(* CODESYS project Discrete.library
   Placeholder: Discrete
   Title: Discrete
   Version: 2025.10.15.1
   Company: Photara

Project tree, tasks and I/O mapping:
  libraries: Base, * (Photara); Tc2_Standard, * (Beckhoff Automation GmbH); Tc2_System, * (Beckhoff Automation GmbH); TcUnit, * (www.tcunit.org)
  DUTs/
    data type E_DiscreteComponentState
    data type E_DiscretePositionType
    data type ST_DiscreteConfiguration
    data type ST_DiscreteStatus
  GVLs/
    global variables GC_Discrete
    global variables GPL_Discrete
  ITFs/
    interface I_DiscreteBase: Activate, Deactivate, P_DiscreteStatus
    interface I_DiscreteBaseConfiguration: P_DiscreteConfiguration
  POUs/
    Actuator/
      GVLs/
        global variables GC_Actuator
        global variables GPL_Actuator
      ITFs/
        interface I_ActuatorBase: Extend, Retract
      function block FB_Actuator [ST]: Extend, Retract, Activate, Deactivate, _SetCommandPermIntlkConfiguration, CyclicLogic
      function block FB_ActuatorFeedback [ST]: _EvaluateCompletionConditions, _InitializeChildrenDependencies, _SetDependencyConfiguration, CyclicLogic
    Tests/
      MockComponents/
        function block FB_TestActuator [ST]: P_TP_CmdConfigurations, P_TP_Commands, P_TP_iControlMode, P_TP_iSystemPermIntlk, P_TP_PermIntlkConfigurations, CyclicLogic
        function block FB_TestActuatorFeedback [ST]: P_I_SensorCfgExt, P_I_SensorCfgRet, P_I_SensorExt, P_I_SensorRet, _InitializeChildrenDependencies, _SetDependencyConfiguration, CyclicLogic
      function block FB_ActuatorBasicTests [ST]: _GetDiscreteComponent, _GetDiscreteComponentConfig
      function block FB_ActuatorFeedbackTests [ST]: _GetDiscreteComponent, _GetDiscreteComponentConfig, Test_FeedbackExtend_CompletesEarlyOnSensor, Test_FeedbackExtend_TimeoutWithoutSensor, Test_FeedbackRetract_CompletesEarlyOnSensor, Test_FeedbackRetract_TimeoutWithoutSensor
      function block FB_DiscreteBaseTests [ST]: _GetDiscreteComponent, _GetDiscreteComponentConfig, Test_ActivateCommandIdempotency, Test_CoilTruthTable_Active, Test_CoilTruthTable_Alternate, Test_CoilTruthTable_BothOn_FaultExpected, Test_CoilTruthTable_Neutral, Test_DeactivateCommandIdempotency, Test_DeviceReportsError_SetsFaultFlagAndOutputsOff, Test_DirectTransition_ActiveToAlternate, Test_DirectTransition_AlternateToActive, Test_ErrorRecovery_ClearsAndReturnsToNeutral, Test_InitializationSetsNeutralStateWithNoOutputs, Test_InvalidCommand_DoesNotChangeOutputs, Test_PermissiveInterlock_BlocksActivation, Test_PermissiveInterlock_BlocksAlternate, Test_RapidStateChanges_EndInExpectedState, Test_StateStabilityAcrossMultipleCycles, Test_ThreePositionDevice_ActivatesAlternateOutputOnly, Test_ThreePositionDevice_ActivatesPrimaryOutputOnly, Test_ThreePositionDevice_DeactivateTurnsOffBothOutputs, Test_ThreePositionDevice_NeverActivatesBothOutputsSimultaneously, Test_TransitionFromActiveToAlternateTurnsOffActiveFirst, Test_TwoPositionDevice_ActivatesCorrectOutput, Test_TwoPositionDevice_DeactivatesAllOutputs, Test_TwoPositionDevice_IgnoresAlternateRequest
      function block FB_ElectrostaticTests [ST]: _GetDiscreteComponent, _GetDiscreteComponentConfig
      function block FB_VacuumPurgeTests [ST]: _GetDiscreteComponent, _GetDiscreteComponentConfig
    function block FB_DiscreteBase [ST]: CyclicLogic, Activate, Deactivate, P_DiscreteConfiguration, P_DiscreteStatus, _InitializeReferences, _SetCommandPermIntlkConfiguration, _Activate, _Deactivate, _EvaluateCompletionConditions, _UpdateComponentStatus
    function block FB_Electrostatic [ST]: Activate, Deactivate, CyclicLogic
    function block FB_VacuumPurge [ST]: Activate, Deactivate, CyclicLogic, Purge, Vacuum
    program MAIN [ST]
    program PRG_TEST [ST]
*)

// DUTs/E_DiscreteComponentState
{attribute 'qualified_only'}
{attribute 'strict'}
{attribute 'to_string'}
TYPE E_DiscreteComponentState :
(
	Indeterminate := 0, //Undefined/Init
	Neutral 	:= 1, //Off/Determined but no output
	Active 		:= 2, //On/Vaccum
	Alternate	:= 3 //Purge
);
END_TYPE

// DUTs/E_DiscretePositionType
{attribute 'qualified_only'}
{attribute 'strict'}
{attribute 'to_string'}
TYPE E_DiscretePositionType  :
(
	TwoPositionDevice := 0,
	ThreePositionDevice := 1
);
END_TYPE

// DUTs/ST_DiscreteConfiguration
TYPE ST_DiscreteConfiguration :
STRUCT
	ComponentConfiguration 	: REFERENCE TO ST_ComponentConfiguration;
	PositionType			: E_DiscretePositionType;
	ActivationDuration		: TIME	:= Tc2_System.Global_Variables.DEFAULT_ADS_TIMEOUT; // assuming no feedback
	DeactivationDuration	: TIME 	:= T#10MS; // assuming no feedback
END_STRUCT
END_TYPE

// DUTs/ST_DiscreteStatus
TYPE ST_DiscreteStatus :
STRUCT
	ComponentStatus 		: REFERENCE TO ST_ComponentStatus;
	BinaryComponentState 	: E_DiscreteComponentState;
	
	PrimaryOutput 	AT %Q*	: BOOL; // ie., Vaccum
	SecondaryOutput	AT %Q*	: BOOL; // ie., Purge
END_STRUCT
END_TYPE

// GVLs/GC_Discrete
{attribute 'qualified_only'}
{attribute 'global_init_slot' := '40615'}
VAR_GLOBAL CONSTANT
	INDEX_COMMAND_MIN 	: DINT := GPL_Discrete.INDEX_COMMAND_MIN;
	INDEX_COMMAND_MAX 	: DINT := GPL_Discrete.INDEX_COMMAND_MAX;
	CMD_VAC				: DINT := 2;
	CMD_PURGE			: DINT := 3;
	CMD_EXTEND			: DINT := 4;
	CMD_RETRACT			: DINT := 5;
	INDEX_TEST_MIN		: DINT := 0;
	INDEX_TEST_MAX		: DINT := 30;
END_VAR

// GVLs/GPL_Discrete
{attribute 'qualified_only'}
{attribute 'global_init_slot' := '40515'}
VAR_GLOBAL CONSTANT
	INDEX_COMMAND_MIN 	: DINT := 0;
	INDEX_COMMAND_MAX 	: DINT := 4;
END_VAR

// POUs/Actuator/GVLs/GC_Actuator
{attribute 'qualified_only'}
{attribute 'global_init_slot' := '40603'}
VAR_GLOBAL CONSTANT
	INDEX_COMMAND_MIN		: DINT := GPL_Actuator.INDEX_COMMAND_MIN;
	INDEX_COMMAND_MAX		: DINT := GPL_Actuator.INDEX_COMMAND_MAX;
	Extend					: DINT := 2;
END_VAR

// POUs/Actuator/GVLs/GPL_Actuator
{attribute 'qualified_only'}
{attribute 'global_init_slot' := '40503'}
VAR_GLOBAL CONSTANT
	INDEX_COMMAND_MIN		: DINT := 0;
	INDEX_COMMAND_MAX		: DINT := 7;
END_VAR

// ITFs/I_DiscreteBase
INTERFACE I_DiscreteBase EXTENDS Base.I_BaseCyclic

METHOD Activate : Base.E_CommandResult
END_METHOD

METHOD Deactivate : Base.E_CommandResult
END_METHOD

PROPERTY P_DiscreteStatus : REFERENCE TO ST_DiscreteStatus
GET
END_GET
END_PROPERTY

END_INTERFACE

// ITFs/I_DiscreteBaseConfiguration
INTERFACE I_DiscreteBaseConfiguration EXTENDS Base.I_BaseCyclic

PROPERTY P_DiscreteConfiguration : REFERENCE TO ST_DiscreteConfiguration
GET
END_GET
END_PROPERTY

END_INTERFACE

// POUs/Actuator/ITFs/I_ActuatorBase
INTERFACE I_ActuatorBase EXTENDS __SYSTEM.IQueryInterface

METHOD Extend : E_CommandResult
VAR_INPUT
END_VAR
END_METHOD

METHOD Retract : E_CommandResult
VAR_INPUT
END_VAR
END_METHOD

END_INTERFACE

// POUs/Actuator/FB_Actuator
{attribute 'no_explicit_call' := 'do not call this POU directly'}
FUNCTION_BLOCK FB_Actuator EXTENDS FB_DiscreteBase IMPLEMENTS I_ActuatorBase
VAR CONSTANT
	// Use base class command indices - no need for separate actuator command indices
	// Extend = Activate (INDEX_CMD_ACTIVATE from base class)
	// Retract = Deactivate (INDEX_CMD_DEACTIVATE from base class)
END_VAR

VAR
	TestPermissiveFalse	: BOOL;
	TestPermissiveTrue	: BOOL := TRUE;
END_VAR

METHOD Extend : E_CommandResult
// Alias for Activate (Extend is the active state)
Extend := Activate();
END_METHOD

METHOD Retract : E_CommandResult
// Alias for Deactivate (Retract is the idle state)
Retract := Deactivate();
END_METHOD

METHOD Activate : Base.E_CommandResult
// Simply call the parent's Activate method - it handles everything
Activate := SUPER^.Activate();
END_METHOD

METHOD Deactivate : Base.E_CommandResult
// Simply call the parent's Deactivate method - it handles everything
Deactivate := SUPER^.Deactivate();
END_METHOD

METHOD PROTECTED _SetCommandPermIntlkConfiguration : BOOL
// Call parent configuration FIRST to set up base commands
SUPER^._SetCommandPermIntlkConfiguration();

//Configure as Two-Position Device
SUPER^.DiscreteComponentConfiguration.PositionType := E_DiscretePositionType.TwoPositionDevice;

//Command Extend
SUPER^.DiscreteComponentConfiguration.ActivationDuration	:= T#20S;
SUPER^.DiscreteComponentConfiguration.DeactivationDuration	:= T#5S;

// Override base command descriptions to use actuator terminology (Extend maps to Activate)
CommandPermIntlkConfiguration[INDEX_CMD_ACTIVATE].P_CommandConfiguration.CommandDescription					:= 'Extend';
CommandPermIntlkConfiguration[INDEX_CMD_ACTIVATE].P_CommandConfiguration.CommandIndex							:= INDEX_CMD_ACTIVATE;
CommandPermIntlkConfiguration[INDEX_CMD_ACTIVATE].P_CommandConfiguration.CommandPOUName						:= 'Extend';
CommandPermIntlkConfiguration[INDEX_CMD_ACTIVATE].P_CommandConfiguration.Priority								:= Base.E_CommandPriority.Priority_Normal;
CommandPermIntlkConfiguration[INDEX_CMD_ACTIVATE].P_CommandConfiguration.TimeoutTime							:= SUPER^.DiscreteComponentConfiguration.ActivationDuration;
CommandPermIntlkConfiguration[INDEX_CMD_ACTIVATE].P_CommandConfiguration.CompletionCondition					REF= SUPER^.CommandCompletionConditions[INDEX_CMD_ACTIVATE];

CommandPermIntlkConfiguration[INDEX_CMD_ACTIVATE].P_CommandConfiguration.PermIntlkConfiguration.PermIntlkObj[0].Condition		REF= TestPermissiveTrue;
CommandPermIntlkConfiguration[INDEX_CMD_ACTIVATE].P_CommandConfiguration.PermIntlkConfiguration.PermIntlkObj[0].Description	:= 'TestPermssiveFalse';
CommandPermIntlkConfiguration[INDEX_CMD_ACTIVATE].P_CommandConfiguration.PermIntlkConfiguration.PermIntlkObj[0].Index	:= 0;

//Command Retract
// Override base command descriptions to use actuator terminology (Retract maps to Deactivate)
CommandPermIntlkConfiguration[INDEX_CMD_DEACTIVATE].P_CommandConfiguration.CommandDescription					:= 'Retract';
CommandPermIntlkConfiguration[INDEX_CMD_DEACTIVATE].P_CommandConfiguration.CommandIndex						:= INDEX_CMD_DEACTIVATE;
CommandPermIntlkConfiguration[INDEX_CMD_DEACTIVATE].P_CommandConfiguration.CommandPOUName						:= 'Retract';
CommandPermIntlkConfiguration[INDEX_CMD_DEACTIVATE].P_CommandConfiguration.Priority							:= Base.E_CommandPriority.Priority_High;
CommandPermIntlkConfiguration[INDEX_CMD_DEACTIVATE].P_CommandConfiguration.TimeoutTime							:= SUPER^.DiscreteComponentConfiguration.DeactivationDuration;
CommandPermIntlkConfiguration[INDEX_CMD_DEACTIVATE].P_CommandConfiguration.CompletionCondition					REF= SUPER^.CommandCompletionConditions[INDEX_CMD_DEACTIVATE];

// CommandPermIntlkConfiguration[INDEX_COMMAND_RETRACT].P_CommandConfiguration.PermIntlkConfiguration.PermIntlkObj[].Condition	:= ;
// CommandPermIntlkConfiguration[INDEX_COMMAND_RETRACT].P_CommandConfiguration.PermIntlkConfiguration.PermIntlkObj[].Description	:= ;
// CommandPermIntlkConfiguration[INDEX_COMMAND_RETRACT].P_CommandConfiguration.PermIntlkConfiguration.PermIntlkObj[].Index	:= ;

_SetCommandPermIntlkConfiguration	:= TRUE;
END_METHOD

METHOD CyclicLogic
SUPER^.CyclicLogic();
END_METHOD

END_FUNCTION_BLOCK

// POUs/FB_DiscreteBase
{attribute 'no_explicit_call' := 'do not call this POU directly'}
FUNCTION_BLOCK ABSTRACT FB_DiscreteBase EXTENDS FB_Component<GC_Discrete.INDEX_COMMAND_MIN, GC_Discrete.INDEX_COMMAND_MAX> IMPLEMENTS I_DiscreteBase, I_DiscreteBaseConfiguration
VAR CONSTANT
	INDEX_CMD_ACTIVATE			: DINT := 0;
	INDEX_CMD_DEACTIVATE 		: DINT := 1;
END_VAR
VAR
	DiscreteComponentConfiguration				: ST_DiscreteConfiguration;
	DiscreteComponentStatus						: ST_DiscreteStatus;
END_VAR

METHOD CyclicLogic
SUPER^.CyclicLogic();
END_METHOD

METHOD Activate : Base.E_CommandResult
ExecuteCommand(CmdIndex := INDEX_CMD_ACTIVATE);

IF SUPER^.iCommands[INDEX_CMD_ACTIVATE].P_CommandStatus.Result = Base.E_CommandResult.Accepted THEN
	_Activate();
END_IF

Activate := SUPER^.iCommands[INDEX_CMD_ACTIVATE].P_CommandStatus.Result;
END_METHOD

METHOD Deactivate : Base.E_CommandResult
ExecuteCommand(CmdIndex := INDEX_CMD_DEACTIVATE);

IF SUPER^.iCommands[INDEX_CMD_DEACTIVATE].P_CommandStatus.Result = Base.E_CommandResult.Accepted THEN
	_Deactivate();
END_IF

Deactivate := SUPER^.iCommands[INDEX_CMD_DEACTIVATE].P_CommandStatus.Result;
END_METHOD

PROPERTY P_DiscreteConfiguration : REFERENCE TO ST_DiscreteConfiguration
GET
P_DiscreteConfiguration REF= DiscreteComponentConfiguration;
END_GET
END_PROPERTY

PROPERTY P_DiscreteStatus : REFERENCE TO ST_DiscreteStatus
GET
P_DiscreteStatus REF= DiscreteComponentStatus;
END_GET
END_PROPERTY

METHOD PROTECTED _InitializeReferences : BOOL
//Initialize data references
//Order is important!
BaseConfiguration.InstancePath 							REF= InstancePath;

ComponentConfiguration.BaseConfiguration 				REF= SUPER^.BaseConfiguration;
                                                    
ComponentStatus.BaseStatus								REF= SUPER^.BaseStatus;

ComponentStatus.AmsNetId								REF= ComponentConfiguration.AmsNetId;
                                                    
DiscreteComponentConfiguration.ComponentConfiguration	REF= SUPER^.ComponentConfiguration;

DiscreteComponentStatus.ComponentStatus					REF= SUPER^.ComponentStatus;

_InitializeReferences				:= TRUE;
END_METHOD

METHOD PROTECTED _SetCommandPermIntlkConfiguration : BOOL
//Command On
CommandPermIntlkConfiguration[INDEX_CMD_ACTIVATE].P_CommandConfiguration.AbortOnInterlockDrop					:= TRUE;
CommandPermIntlkConfiguration[INDEX_CMD_ACTIVATE].P_CommandConfiguration.CommandDescription						:= 'Activate';
CommandPermIntlkConfiguration[INDEX_CMD_ACTIVATE].P_CommandConfiguration.CommandIndex							:= INDEX_CMD_ACTIVATE;
CommandPermIntlkConfiguration[INDEX_CMD_ACTIVATE].P_CommandConfiguration.CommandPOUName							:= 'Activate';
//CommandPermIntlkConfiguration[INDEX_CMD_ACTIVATE].P_CommandConfiguration.PermIntlkConfiguredAsInterlock		:= TRUE;
CommandPermIntlkConfiguration[INDEX_CMD_ACTIVATE].P_CommandConfiguration.Priority								:= Base.E_CommandPriority.Priority_Normal;
CommandPermIntlkConfiguration[INDEX_CMD_ACTIVATE].P_CommandConfiguration.CompletionCondition					REF= SUPER^.CommandCompletionConditions[INDEX_CMD_ACTIVATE];
//CommandPermIntlkConfiguration[INDEX_CMD_ACTIVATE].P_CommandConfiguration.TimeoutTime							:= DiscreteComponentConfiguration.ActivationDuration;

// CommandPermIntlkConfiguration[INDEX_CMD_ACTIVATE].P_CommandConfiguration.PermIntlkConfiguration.PermIntlkObj[].Condition	:= ;
// CommandPermIntlkConfiguration[INDEX_CMD_ACTIVATE].P_CommandConfiguration.PermIntlkConfiguration.PermIntlkObj[].Description	:= ;
// CommandPermIntlkConfiguration[INDEX_CMD_ACTIVATE].P_CommandConfiguration.PermIntlkConfiguration.PermIntlkObj[].Index	:= ;

//Command Off
//CommandPermIntlkConfiguration[INDEX_CMD_DEACTIVATE].P_CommandConfiguration.AbortOnInterlockDrop				:= TRUE;
CommandPermIntlkConfiguration[INDEX_CMD_DEACTIVATE].P_CommandConfiguration.CommandDescription					:= 'Deactivate';
CommandPermIntlkConfiguration[INDEX_CMD_DEACTIVATE].P_CommandConfiguration.CommandIndex							:= INDEX_CMD_DEACTIVATE;
CommandPermIntlkConfiguration[INDEX_CMD_DEACTIVATE].P_CommandConfiguration.CommandPOUName						:= 'Deactivate';
//CommandPermIntlkConfiguration[INDEX_CMD_DEACTIVATE].P_CommandConfiguration.PermIntlkConfiguredAsInterlock		:= TRUE;
CommandPermIntlkConfiguration[INDEX_CMD_DEACTIVATE].P_CommandConfiguration.Priority								:= Base.E_CommandPriority.Priority_High;
CommandPermIntlkConfiguration[INDEX_CMD_DEACTIVATE].P_CommandConfiguration.TimeoutTime							:= DiscreteComponentConfiguration.DeactivationDuration;
CommandPermIntlkConfiguration[INDEX_CMD_DEACTIVATE].P_CommandConfiguration.CompletionCondition					REF= SUPER^.CommandCompletionConditions[INDEX_CMD_DEACTIVATE];
CommandPermIntlkConfiguration[INDEX_CMD_DEACTIVATE].P_CommandConfiguration.TimeoutTime							:= DiscreteComponentConfiguration.DeactivationDuration;

// CommandPermIntlkConfiguration[INDEX_CMD_DEACTIVATE].P_CommandConfiguration.PermIntlkConfiguration.PermIntlkObj[].Condition	:= ;
// CommandPermIntlkConfiguration[INDEX_CMD_DEACTIVATE].P_CommandConfiguration.PermIntlkConfiguration.PermIntlkObj[].Description	:= ;
// CommandPermIntlkConfiguration[INDEX_CMD_DEACTIVATE].P_CommandConfiguration.PermIntlkConfiguration.PermIntlkObj[].Index	:= ;

_SetCommandPermIntlkConfiguration	:= TRUE;
END_METHOD

METHOD PROTECTED _Activate
// Continuous mode: Hold output ON while command is busy
DiscreteComponentStatus.PrimaryOutput := TRUE;
DiscreteComponentStatus.SecondaryOutput := FALSE; // Safety: ensure alternate is off
END_METHOD

METHOD PROTECTED _Deactivate
// Continuous mode: Hold output OFF while command is busy
DiscreteComponentStatus.PrimaryOutput := FALSE;
DiscreteComponentStatus.SecondaryOutput := FALSE; // Safety: ensure alternate is off
END_METHOD

METHOD PROTECTED _EvaluateCompletionConditions : BOOL
// Set default completion conditions - commands complete immediately after output transition
// Derived classes can override to use different completion criteria (timeout, sensor feedback, etc.)
SUPER^.CommandCompletionConditions[INDEX_CMD_ACTIVATE]            		:= (DiscreteComponentStatus.PrimaryOutput AND NOT DiscreteComponentStatus.SecondaryOutput);
SUPER^.CommandCompletionConditions[INDEX_CMD_DEACTIVATE]            	:= (NOT DiscreteComponentStatus.PrimaryOutput AND NOT DiscreteComponentStatus.SecondaryOutput);

// Call generic logging implementation
_EvaluateCompletionConditions := TRUE;
END_METHOD

METHOD PROTECTED _UpdateComponentStatus: Base.I_ComponentFull
// Check configuration for device type
IF DiscreteComponentConfiguration.PositionType = E_DiscretePositionType.TwoPositionDevice THEN
	// Two-position device: Secondary output is always FALSE
	// Only two states are valid: Active and Neutral
	DiscreteComponentStatus.SecondaryOutput := FALSE;

	// Update state based on primary output only
	IF DiscreteComponentStatus.PrimaryOutput THEN
		// Primary output active = Active state
		DiscreteComponentStatus.BinaryComponentState := E_DiscreteComponentState.Active;
	ELSE
		// Primary output inactive = Neutral state
		DiscreteComponentStatus.BinaryComponentState := E_DiscreteComponentState.Neutral;
	END_IF
ELSE
	// Three-position device: Support all three states
	// Update component state based on primary and secondary outputs
	IF DiscreteComponentStatus.SecondaryOutput THEN
		// Secondary output active = Alternate state (e.g., Purge)
		DiscreteComponentStatus.BinaryComponentState := E_DiscreteComponentState.Alternate;
	ELSIF DiscreteComponentStatus.PrimaryOutput THEN
		// Primary output active, secondary inactive = Active state (e.g., Vacuum)
		DiscreteComponentStatus.BinaryComponentState := E_DiscreteComponentState.Active;
	ELSIF NOT DiscreteComponentStatus.PrimaryOutput AND NOT DiscreteComponentStatus.SecondaryOutput THEN
		// Both outputs inactive = Neutral state (Off)
		DiscreteComponentStatus.BinaryComponentState := E_DiscreteComponentState.Neutral;
	ELSE
		// Should not reach here, but if we do = Indeterminate
		DiscreteComponentStatus.BinaryComponentState := E_DiscreteComponentState.Indeterminate;
	END_IF
END_IF

_UpdateComponentStatus := THIS^;
END_METHOD

END_FUNCTION_BLOCK

// POUs/Actuator/FB_ActuatorFeedback
{attribute 'no_explicit_call' := 'do not call this POU directly'}
FUNCTION_BLOCK FB_ActuatorFeedback EXTENDS FB_Actuator
VAR
	SensorFeedbackExtended		: Base.FB_Debounce;
	SensorFeedbackRetracted		: Base.FB_Debounce;
	iDebounceExt				: Base.I_Debounce	:= SensorFeedbackExtended;
	iDebounceRet				: Base.I_Debounce	:= SensorFeedbackRetracted;
END_VAR

METHOD PROTECTED _EvaluateCompletionConditions : BOOL
// Set feedback-specific completion conditions - commands complete when sensors confirm position
IF iDebounceExt <> 0 THEN
	SUPER^.CommandCompletionConditions[INDEX_CMD_ACTIVATE]            	:= iDebounceExt.P_DebounceStatus.DebouncedSignal;
END_IF

IF iDebounceRet <> 0 THEN
	SUPER^.CommandCompletionConditions[INDEX_CMD_DEACTIVATE]            	:= iDebounceRet.P_DebounceStatus.DebouncedSignal;
END_IF

// Call base class logging method
_EvaluateCompletionConditions := TRUE;
END_METHOD

METHOD PROTECTED _InitializeChildrenDependencies : BOOL
// Initialize concrete configurations and wire directly to Commands
FOR CommandIndexCyclic := LOWER_BOUND(Commands,1) TO UPPER_BOUND(Commands,1) BY 1 DO

	// Inject configurations directly - TwinCAT auto-converts to interfaces
	Commands[CommandIndexCyclic].InjectConfigurations(
		iComponent := THIS^,
		iCommandConfiguration := CommandPermIntlkConfiguration[CommandIndexCyclic],
		iPermIntlkConfiguration := CommandPermIntlkConfiguration[CommandIndexCyclic]);
		
	CommandPermIntlkConfiguration[CommandIndexCyclic].Initialize();
	Commands[CommandIndexCyclic].Initialize();
END_FOR

CommandBuffer.Initialize();

fbHashDJB2_PouName.Initialize();
HashTablePouName.Initialize();

SensorFeedbackExtended.Initialize();
SensorFeedbackRetracted.Initialize();

HashTablePouName.InjectHashFunction(iHashFunction := iHashDJB2_PouName);

_InitializeChildrenDependencies := TRUE;
END_METHOD

METHOD PROTECTED _SetDependencyConfiguration : BOOL
SensorFeedbackExtended.P_DebounceConfiguration.BaseConfiguration.InSimulation	:= TRUE;
SensorFeedbackRetracted.P_DebounceConfiguration.BaseConfiguration.InSimulation	:= TRUE;
SensorFeedbackExtended.P_DebounceConfiguration.tOnDelay		:= T#50MS;
SensorFeedbackExtended.P_DebounceConfiguration.tOffDelay	:= T#50MS;

_SetDependencyConfiguration	:= TRUE;
END_METHOD

METHOD CyclicLogic
SUPER^.CyclicLogic();

SensorFeedbackExtended.CyclicLogic();
SensorFeedbackRetracted.CyclicLogic();
END_METHOD

END_FUNCTION_BLOCK

// POUs/Tests/MockComponents/FB_TestActuator
FUNCTION_BLOCK FB_TestActuator EXTENDS FB_Actuator
VAR_INPUT
END_VAR
VAR_OUTPUT
END_VAR
VAR
END_VAR

PROPERTY P_TP_CmdConfigurations : REFERENCE TO ARRAY[MinIndexComponentCmd..MaxIndexComponentCmd] OF FB_CmdPermIntlkConfiguration
GET
P_TP_CmdConfigurations REF= SUPER^.CommandPermIntlkConfiguration;
END_GET
END_PROPERTY

PROPERTY P_TP_Commands : REFERENCE TO ARRAY[MinIndexComponentCmd..MaxIndexComponentCmd] OF FB_Command
GET
P_TP_Commands REF= SUPER^.Commands;
END_GET
END_PROPERTY

PROPERTY P_TP_iControlMode : REFERENCE TO I_ControlMode
GET
P_TP_iControlMode REF= SUPER^._ControlMode;
END_GET
END_PROPERTY

PROPERTY P_TP_iSystemPermIntlk : REFERENCE TO I_PermIntlk
GET
P_TP_iSystemPermIntlk REF= SUPER^._SystemPermIntlk;
END_GET
END_PROPERTY

PROPERTY P_TP_PermIntlkConfigurations : REFERENCE TO ARRAY[MinIndexComponentCmd..MaxIndexComponentCmd] OF FB_CmdPermIntlkConfiguration
GET
P_TP_PermIntlkConfigurations REF= SUPER^.CommandPermIntlkConfiguration;
END_GET
END_PROPERTY

METHOD CyclicLogic
SUPER^.CyclicLogic();
END_METHOD

END_FUNCTION_BLOCK

// POUs/Tests/MockComponents/FB_TestActuatorFeedback
{attribute 'no_explicit_call' := 'do not call this POU directly'}
FUNCTION_BLOCK FB_TestActuatorFeedback EXTENDS FB_TestActuator
VAR
	SensorFeedbackExtended		: Base.FB_Debounce;
	SensorFeedbackRetracted		: Base.FB_Debounce;
	iDebounceExt				: Base.I_Debounce				:= SensorFeedbackExtended;
	iDebounceRet				: Base.I_Debounce				:= SensorFeedbackRetracted;
	iDebounceConfigExt			: Base.I_DebounceConfiguration	:= SensorFeedbackExtended;
	iDebounceConfigRet			: Base.I_DebounceConfiguration  := SensorFeedbackRetracted;
END_VAR

PROPERTY P_I_SensorCfgExt : REFERENCE TO Base.I_DebounceConfiguration
GET
P_I_SensorCfgExt REF= iDebounceConfigExt;
END_GET
END_PROPERTY

PROPERTY P_I_SensorCfgRet : REFERENCE TO Base.I_DebounceConfiguration
GET
P_I_SensorCfgRet REF= iDebounceConfigRet;
END_GET
END_PROPERTY

PROPERTY P_I_SensorExt : REFERENCE TO Base.I_Debounce
GET
P_I_SensorExt REF= iDebounceExt;
END_GET
END_PROPERTY

PROPERTY P_I_SensorRet : REFERENCE TO Base.I_Debounce
GET
P_I_SensorRet REF= iDebounceRet;
END_GET
END_PROPERTY

METHOD PROTECTED _InitializeChildrenDependencies : BOOL
// Initialize concrete configurations and wire directly to Commands
FOR CommandIndexCyclic := LOWER_BOUND(Commands,1) TO UPPER_BOUND(Commands,1) BY 1 DO

	// Inject configurations directly - TwinCAT auto-converts to interfaces
	Commands[CommandIndexCyclic].InjectConfigurations(
		iComponent := THIS^,
		iCommandConfiguration := CommandPermIntlkConfiguration[CommandIndexCyclic],
		iPermIntlkConfiguration := CommandPermIntlkConfiguration[CommandIndexCyclic]);
		
	CommandPermIntlkConfiguration[CommandIndexCyclic].Initialize();
	Commands[CommandIndexCyclic].Initialize();
END_FOR

CommandBuffer.Initialize();

fbHashDJB2_PouName.Initialize();
HashTablePouName.Initialize();

SensorFeedbackExtended.Initialize();
SensorFeedbackRetracted.Initialize();

HashTablePouName.InjectHashFunction(iHashFunction := iHashDJB2_PouName);

_InitializeChildrenDependencies := TRUE;
END_METHOD

METHOD PROTECTED _SetDependencyConfiguration : BOOL
SensorFeedbackExtended.P_DebounceConfiguration.BaseConfiguration.InSimulation	:= TRUE;
SensorFeedbackRetracted.P_DebounceConfiguration.BaseConfiguration.InSimulation	:= TRUE;
SensorFeedbackExtended.P_DebounceConfiguration.tOnDelay		:= T#50MS;
SensorFeedbackExtended.P_DebounceConfiguration.tOffDelay	:= T#50MS;

_SetDependencyConfiguration	:= TRUE;
END_METHOD

METHOD CyclicLogic
SUPER^.CyclicLogic();

SensorFeedbackExtended.CyclicLogic();
SensorFeedbackRetracted.CyclicLogic();
END_METHOD

END_FUNCTION_BLOCK

// POUs/Tests/FB_ActuatorBasicTests
FUNCTION_BLOCK FB_ActuatorBasicTests EXTENDS FB_DiscreteBaseTests

VAR
	afbActuator			: ARRAY[GC_Discrete.INDEX_TEST_MIN..GC_Discrete.INDEX_TEST_MAX] OF FB_TestActuator;
END_VAR

// All test methods are inherited from FB_DiscreteBaseTests
SUPER^();

METHOD PROTECTED _GetDiscreteComponent : I_DiscreteBase
VAR_INPUT
	Index : DINT;
END_VAR
// Return the actuator instance at the given index
_GetDiscreteComponent := afbActuator[Index];
END_METHOD

METHOD PROTECTED _GetDiscreteComponentConfig : I_DiscreteBaseConfiguration
VAR_INPUT
	Index : DINT;
END_VAR
// Return the actuator instance at the given index as configuration interface
_GetDiscreteComponentConfig := afbActuator[Index];
END_METHOD

END_FUNCTION_BLOCK

// POUs/Tests/FB_DiscreteBaseTests
FUNCTION_BLOCK ABSTRACT FB_DiscreteBaseTests EXTENDS TcUnit.FB_TestSuite

VAR
	iDiscreteComponent 	: I_DiscreteBase;
	iDiscreteConfig		: I_DiscreteBaseConfiguration;
	i 					: INT;
END_VAR
VAR CONSTANT
	// Core merged test indices
	INDEX_INITIALIZATION				: DINT := 0;
	INDEX_ACTIVATE_IDEMPOTENCY			: DINT := 1;
	INDEX_DEACTIVATE_IDEMPOTENCY		: DINT := 2;
	INDEX_STATE_STABILITY				: DINT := 3;

	// Safety test indices
	INDEX_NEVER_BOTH_OUTPUTS			: DINT := 4;
	INDEX_COIL_BOTH_ON_FAULT			: DINT := 5;
	INDEX_BREAK_BEFORE_MAKE				: DINT := 6;

	// Truth table test indices
	INDEX_COIL_NEUTRAL					: DINT := 7;
	INDEX_COIL_ACTIVE					: DINT := 8;
	INDEX_COIL_ALTERNATE				: DINT := 9;

	// Two-position device test indices
	INDEX_TWO_POS_ACTIVATE				: DINT := 10;
	INDEX_TWO_POS_DEACTIVATE			: DINT := 11;
	INDEX_TWO_POS_IGNORE_ALT			: DINT := 12;

	// Three-position device test indices
	INDEX_THREE_POS_PRIMARY				: DINT := 13;
	INDEX_THREE_POS_ALTERNATE			: DINT := 14;
	INDEX_THREE_POS_DEACTIVATE			: DINT := 15;

	// State transition test indices
	INDEX_ACTIVE_TO_ALTERNATE			: DINT := 16;
	INDEX_ALTERNATE_TO_ACTIVE			: DINT := 17;
	INDEX_RAPID_STATE_CHANGES			: DINT := 18;

	// Error handling test indices
	INDEX_INVALID_COMMAND				: DINT := 19;
	INDEX_DEVICE_ERROR					: DINT := 20;
	INDEX_ERROR_RECOVERY				: DINT := 21;

	// Interlock test indices
	INDEX_INTERLOCK_ACTIVATION			: DINT := 22;
	INDEX_INTERLOCK_ALTERNATE			: DINT := 23;

	// Reserve index 24 for future use
	INDEX_RESERVED						: DINT := 24;
END_VAR

// Core Safety Tests
Test_ThreePositionDevice_NeverActivatesBothOutputsSimultaneously();
Test_CoilTruthTable_BothOn_FaultExpected();
Test_TransitionFromActiveToAlternateTurnsOffActiveFirst();

// Truth Table Validation
Test_CoilTruthTable_Neutral();
Test_CoilTruthTable_Active();
Test_CoilTruthTable_Alternate();

// Merged Core State Tests
Test_InitializationSetsNeutralStateWithNoOutputs();
Test_ActivateCommandIdempotency();
Test_DeactivateCommandIdempotency();
Test_StateStabilityAcrossMultipleCycles();

// Two-Position Device Tests
Test_TwoPositionDevice_ActivatesCorrectOutput();
Test_TwoPositionDevice_DeactivatesAllOutputs();
Test_TwoPositionDevice_IgnoresAlternateRequest();

// Three-Position Device Tests
Test_ThreePositionDevice_ActivatesPrimaryOutputOnly();
Test_ThreePositionDevice_ActivatesAlternateOutputOnly();
Test_ThreePositionDevice_DeactivateTurnsOffBothOutputs();

// State Transition Tests
Test_DirectTransition_ActiveToAlternate();
Test_DirectTransition_AlternateToActive();
Test_RapidStateChanges_EndInExpectedState();

// Error Handling Tests
Test_InvalidCommand_DoesNotChangeOutputs();
Test_DeviceReportsError_SetsFaultFlagAndOutputsOff();
Test_ErrorRecovery_ClearsAndReturnsToNeutral();

// Interlock Tests
Test_PermissiveInterlock_BlocksActivation();
Test_PermissiveInterlock_BlocksAlternate();

METHOD PROTECTED ABSTRACT _GetDiscreteComponent : I_DiscreteBase
VAR_INPUT
	Index : DINT;
END_VAR
// Abstract method - must be implemented by derived test classes
// Returns the discrete component instance at the given test index
END_METHOD

METHOD PROTECTED ABSTRACT _GetDiscreteComponentConfig : I_DiscreteBaseConfiguration
VAR_INPUT
	Index : DINT;
END_VAR
// Abstract method - must be implemented by derived test classes
// Returns the discrete component instance at the given test index as configuration interface
END_METHOD

METHOD PRIVATE Test_ActivateCommandIdempotency
TEST(__POUNAME());

iDiscreteComponent := _GetDiscreteComponent(INDEX_ACTIVATE_IDEMPOTENCY);
IF iDiscreteComponent = 0 THEN RETURN; END_IF
iDiscreteComponent.CyclicLogic();

// Start from neutral state
iDiscreteComponent.Deactivate();
iDiscreteComponent.CyclicLogic();

AssertEquals_INT(
	Expected := TO_INT(E_DiscreteComponentState.Neutral),
	Actual := TO_INT(iDiscreteComponent.P_DiscreteStatus.BinaryComponentState),
	Message := 'Expected: Neutral starting state'
);

// First activation
iDiscreteComponent.Activate();
iDiscreteComponent.CyclicLogic();

AssertEquals_INT(
	Expected := TO_INT(E_DiscreteComponentState.Active),
	Actual := TO_INT(iDiscreteComponent.P_DiscreteStatus.BinaryComponentState),
	Message := 'Expected: Active state after first activation'
);

AssertTrue(
	Condition := iDiscreteComponent.P_DiscreteStatus.PrimaryOutput,
	Message := 'Primary output should be TRUE after activation'
);

// Second activation (idempotency test)
iDiscreteComponent.Activate();
iDiscreteComponent.CyclicLogic();

AssertEquals_INT(
	Expected := TO_INT(E_DiscreteComponentState.Active),
	Actual := TO_INT(iDiscreteComponent.P_DiscreteStatus.BinaryComponentState),
	Message := 'Expected: Active state unchanged after double activation'
);

AssertTrue(
	Condition := iDiscreteComponent.P_DiscreteStatus.PrimaryOutput,
	Message := 'Primary output should remain TRUE after double activation'
);

TEST_FINISHED();
END_METHOD

METHOD PRIVATE Test_CoilTruthTable_Active
TEST(__POUNAME());

iDiscreteComponent := _GetDiscreteComponent(INDEX_COIL_ACTIVE);
IF iDiscreteComponent = 0 THEN RETURN; END_IF
iDiscreteComponent.CyclicLogic();

// Truth Table: Active State
// Primary Output: TRUE
// Secondary Output: FALSE
// Expected State: Active

// Activate the component
iDiscreteComponent.Activate();
iDiscreteComponent.CyclicLogic();

AssertTrue(
	Condition := iDiscreteComponent.P_DiscreteStatus.PrimaryOutput,
	Message := 'Primary output should be TRUE in Active state'
);

AssertFalse(
	Condition := iDiscreteComponent.P_DiscreteStatus.SecondaryOutput,
	Message := 'Secondary output should be FALSE in Active state'
);

AssertEquals_INT(
	Expected := TO_INT(E_DiscreteComponentState.Active),
	Actual := TO_INT(iDiscreteComponent.P_DiscreteStatus.BinaryComponentState),
	Message := 'Truth table: TRUE/FALSE should result in Active state'
);

// Verify the state remains stable
iDiscreteComponent.CyclicLogic();
iDiscreteComponent.CyclicLogic();

AssertEquals_INT(
	Expected := TO_INT(E_DiscreteComponentState.Active),
	Actual := TO_INT(iDiscreteComponent.P_DiscreteStatus.BinaryComponentState),
	Message := 'Active state should remain stable across cycles'
);

// Manually set outputs to verify truth table
iDiscreteComponent.P_DiscreteStatus.PrimaryOutput := TRUE;
iDiscreteComponent.P_DiscreteStatus.SecondaryOutput := FALSE;
iDiscreteComponent.CyclicLogic();

AssertEquals_INT(
	Expected := TO_INT(E_DiscreteComponentState.Active),
	Actual := TO_INT(iDiscreteComponent.P_DiscreteStatus.BinaryComponentState),
	Message := 'Manual truth table verification: TRUE/FALSE = Active'
);

TEST_FINISHED();
END_METHOD

METHOD PRIVATE Test_CoilTruthTable_Alternate
TEST(__POUNAME());

iDiscreteComponent := _GetDiscreteComponent(INDEX_COIL_ALTERNATE);
IF iDiscreteComponent = 0 THEN RETURN; END_IF
iDiscreteConfig := _GetDiscreteComponentConfig(INDEX_COIL_ALTERNATE);  // Same instance, different interface

// Skip this test for two-position devices
IF iDiscreteConfig.P_DiscreteConfiguration.PositionType = E_DiscretePositionType.TwoPositionDevice THEN
	TEST_FINISHED();
	RETURN;
END_IF

iDiscreteComponent.CyclicLogic();

// Truth Table: Alternate State
// Primary Output: FALSE
// Secondary Output: TRUE
// Expected State: Alternate (e.g., Purge mode)

// Since we don't have an Alternate command yet, manually set the outputs
iDiscreteComponent.P_DiscreteStatus.PrimaryOutput := FALSE;
iDiscreteComponent.P_DiscreteStatus.SecondaryOutput := TRUE;
iDiscreteComponent.CyclicLogic();

AssertFalse(
	Condition := iDiscreteComponent.P_DiscreteStatus.PrimaryOutput,
	Message := 'Primary output should be FALSE in Alternate state'
);

AssertTrue(
	Condition := iDiscreteComponent.P_DiscreteStatus.SecondaryOutput,
	Message := 'Secondary output should be TRUE in Alternate state'
);

AssertEquals_INT(
	Expected := TO_INT(E_DiscreteComponentState.Alternate),
	Actual := TO_INT(iDiscreteComponent.P_DiscreteStatus.BinaryComponentState),
	Message := 'Truth table: FALSE/TRUE should result in Alternate state'
);

// Verify the state remains stable
iDiscreteComponent.CyclicLogic();
iDiscreteComponent.CyclicLogic();

AssertEquals_INT(
	Expected := TO_INT(E_DiscreteComponentState.Alternate),
	Actual := TO_INT(iDiscreteComponent.P_DiscreteStatus.BinaryComponentState),
	Message := 'Alternate state should remain stable across cycles'
);

// Verify outputs remain correct
AssertFalse(
	Condition := iDiscreteComponent.P_DiscreteStatus.PrimaryOutput,
	Message := 'Primary must stay OFF in Alternate state'
);

AssertTrue(
	Condition := iDiscreteComponent.P_DiscreteStatus.SecondaryOutput,
	Message := 'Secondary must stay ON in Alternate state'
);

TEST_FINISHED();
END_METHOD

METHOD PRIVATE Test_CoilTruthTable_BothOn_FaultExpected
TEST(__POUNAME());

iDiscreteComponent := _GetDiscreteComponent(INDEX_COIL_BOTH_ON_FAULT);
IF iDiscreteComponent = 0 THEN RETURN; END_IF
iDiscreteConfig := _GetDiscreteComponentConfig(INDEX_COIL_BOTH_ON_FAULT);  // Same instance, different interface

// Skip this test for two-position devices
IF iDiscreteConfig.P_DiscreteConfiguration.PositionType = E_DiscretePositionType.TwoPositionDevice THEN
	TEST_FINISHED();
	RETURN;
END_IF

iDiscreteComponent.CyclicLogic();

// Truth table test: Both coils ON (fault condition)
// This should never occur in normal operation - indicates hardware/software fault
iDiscreteComponent.P_DiscreteStatus.PrimaryOutput := TRUE;
iDiscreteComponent.P_DiscreteStatus.SecondaryOutput := TRUE;
iDiscreteComponent.CyclicLogic();

// Per our implementation, secondary (Alternate) takes priority when both are on
// This ensures deterministic behavior even in fault conditions
AssertEquals_INT(
	Expected := TO_INT(E_DiscreteComponentState.Alternate),
	Actual := TO_INT(iDiscreteComponent.P_DiscreteStatus.BinaryComponentState),
	Message := 'Both outputs ON should result in Alternate state (secondary priority)'
);

// In a production system, this condition should also:
// 1. Set an error/fault flag
// 2. Log the fault condition
// 3. Potentially trigger a safe shutdown sequence
// These features would need to be implemented in the component

// Test that we can recover from this fault condition
// Manually clear outputs to simulate recovery (until command system is configured)
iDiscreteComponent.P_DiscreteStatus.PrimaryOutput := FALSE;
iDiscreteComponent.P_DiscreteStatus.SecondaryOutput := FALSE;
iDiscreteComponent.CyclicLogic();

AssertEquals_INT(
	Expected := TO_INT(E_DiscreteComponentState.Neutral),
	Actual := TO_INT(iDiscreteComponent.P_DiscreteStatus.BinaryComponentState),
	Message := 'Should be able to recover to Neutral state after fault condition'
);

AssertFalse(
	Condition := iDiscreteComponent.P_DiscreteStatus.PrimaryOutput,
	Message := 'Primary output should be cleared after deactivation'
);

AssertFalse(
	Condition := iDiscreteComponent.P_DiscreteStatus.SecondaryOutput,
	Message := 'Secondary output should be cleared after deactivation'
);

TEST_FINISHED();
END_METHOD

METHOD PRIVATE Test_CoilTruthTable_Neutral
TEST(__POUNAME());

iDiscreteComponent := _GetDiscreteComponent(INDEX_COIL_NEUTRAL);
IF iDiscreteComponent = 0 THEN RETURN; END_IF
iDiscreteComponent.CyclicLogic();

// Truth Table: Neutral State
// Primary Output: FALSE
// Secondary Output: FALSE
// Expected State: Neutral

// Ensure we're starting in neutral state (post-initialization)
AssertFalse(
	Condition := iDiscreteComponent.P_DiscreteStatus.PrimaryOutput,
	Message := 'Primary output should be FALSE in Neutral state'
);

AssertFalse(
	Condition := iDiscreteComponent.P_DiscreteStatus.SecondaryOutput,
	Message := 'Secondary output should be FALSE in Neutral state'
);

AssertEquals_INT(
	Expected := TO_INT(E_DiscreteComponentState.Neutral),
	Actual := TO_INT(iDiscreteComponent.P_DiscreteStatus.BinaryComponentState),
	Message := 'Truth table: FALSE/FALSE should result in Neutral state'
);

// Test deactivate command maintains neutral state
iDiscreteComponent.Deactivate();
iDiscreteComponent.CyclicLogic();

AssertEquals_INT(
	Expected := TO_INT(E_DiscreteComponentState.Neutral),
	Actual := TO_INT(iDiscreteComponent.P_DiscreteStatus.BinaryComponentState),
	Message := 'Deactivate in Neutral state should maintain Neutral'
);

// Test that neutral is the safe/default state
// After any error or unknown condition, system should return to neutral
iDiscreteComponent.P_DiscreteStatus.PrimaryOutput := FALSE;
iDiscreteComponent.P_DiscreteStatus.SecondaryOutput := FALSE;
iDiscreteComponent.CyclicLogic();

AssertEquals_INT(
	Expected := TO_INT(E_DiscreteComponentState.Neutral),
	Actual := TO_INT(iDiscreteComponent.P_DiscreteStatus.BinaryComponentState),
	Message := 'Neutral is the safe default state when both outputs are off'
);

TEST_FINISHED();
END_METHOD

METHOD PRIVATE Test_DeactivateCommandIdempotency
TEST(__POUNAME());

iDiscreteComponent := _GetDiscreteComponent(INDEX_DEACTIVATE_IDEMPOTENCY);
IF iDiscreteComponent = 0 THEN RETURN; END_IF
iDiscreteComponent.CyclicLogic();

// Start from active state
iDiscreteComponent.Activate();
iDiscreteComponent.CyclicLogic();

AssertEquals_INT(
	Expected := TO_INT(E_DiscreteComponentState.Active),
	Actual := TO_INT(iDiscreteComponent.P_DiscreteStatus.BinaryComponentState),
	Message := 'Expected: Active starting state'
);

// First deactivation
iDiscreteComponent.Deactivate();
iDiscreteComponent.CyclicLogic();

AssertEquals_INT(
	Expected := TO_INT(E_DiscreteComponentState.Neutral),
	Actual := TO_INT(iDiscreteComponent.P_DiscreteStatus.BinaryComponentState),
	Message := 'Expected: Neutral state after first deactivation'
);

AssertFalse(
	Condition := iDiscreteComponent.P_DiscreteStatus.PrimaryOutput,
	Message := 'Primary output should be FALSE after deactivation'
);

AssertFalse(
	Condition := iDiscreteComponent.P_DiscreteStatus.SecondaryOutput,
	Message := 'Secondary output should be FALSE after deactivation'
);

// Second deactivation (idempotency test)
iDiscreteComponent.Deactivate();
iDiscreteComponent.CyclicLogic();

AssertEquals_INT(
	Expected := TO_INT(E_DiscreteComponentState.Neutral),
	Actual := TO_INT(iDiscreteComponent.P_DiscreteStatus.BinaryComponentState),
	Message := 'Expected: Neutral state unchanged after double deactivation'
);

AssertFalse(
	Condition := iDiscreteComponent.P_DiscreteStatus.PrimaryOutput,
	Message := 'Primary output should remain FALSE after double deactivation'
);

TEST_FINISHED();
END_METHOD

METHOD PRIVATE Test_DeviceReportsError_SetsFaultFlagAndOutputsOff
TEST(__POUNAME());

iDiscreteComponent := _GetDiscreteComponent(INDEX_DEVICE_ERROR);
IF iDiscreteComponent = 0 THEN RETURN; END_IF
iDiscreteComponent.CyclicLogic();

// Start in Active state
iDiscreteComponent.Activate();
iDiscreteComponent.CyclicLogic();

// TODO: Implement error/fault handling in the component
// When implemented, should:
// 1. Set error flag in component status
// 2. Turn off all outputs for safety
// 3. Log the error
// 4. Possibly require reset before normal operation

// For now, test that Deactivate provides safe shutdown
iDiscreteComponent.Deactivate();
iDiscreteComponent.CyclicLogic();

AssertFalse(
	Condition := iDiscreteComponent.P_DiscreteStatus.PrimaryOutput,
	Message := 'Primary output should be OFF in error/safe state'
);

AssertFalse(
	Condition := iDiscreteComponent.P_DiscreteStatus.SecondaryOutput,
	Message := 'Secondary output should be OFF in error/safe state'
);

AssertEquals_INT(
	Expected := TO_INT(E_DiscreteComponentState.Neutral),
	Actual := TO_INT(iDiscreteComponent.P_DiscreteStatus.BinaryComponentState),
	Message := 'Component should go to safe Neutral state on error'
);

// TODO: Implement full error handling
TEST_FINISHED();
END_METHOD

METHOD PRIVATE Test_DirectTransition_ActiveToAlternate
TEST(__POUNAME());

iDiscreteComponent := _GetDiscreteComponent(INDEX_ACTIVE_TO_ALTERNATE);
IF iDiscreteComponent = 0 THEN RETURN; END_IF
iDiscreteConfig := _GetDiscreteComponentConfig(INDEX_ACTIVE_TO_ALTERNATE);  // Same instance, different interface

// Skip this test for two-position devices
IF iDiscreteConfig.P_DiscreteConfiguration.PositionType = E_DiscretePositionType.TwoPositionDevice THEN
	TEST_FINISHED();
	RETURN;
END_IF

iDiscreteComponent.CyclicLogic();

// Start in Active state
iDiscreteComponent.Activate();
iDiscreteComponent.CyclicLogic();

AssertEquals_INT(
	Expected := TO_INT(E_DiscreteComponentState.Active),
	Actual := TO_INT(iDiscreteComponent.P_DiscreteStatus.BinaryComponentState),
	Message := 'Should start in Active state'
);

// TODO: Implement alternate command when available
// For now, manually set the secondary output to test the state logic
iDiscreteComponent.P_DiscreteStatus.SecondaryOutput := TRUE;
iDiscreteComponent.P_DiscreteStatus.PrimaryOutput := FALSE;
iDiscreteComponent.CyclicLogic();

AssertEquals_INT(
	Expected := TO_INT(E_DiscreteComponentState.Alternate),
	Actual := TO_INT(iDiscreteComponent.P_DiscreteStatus.BinaryComponentState),
	Message := 'Should transition to Alternate state'
);

// Verify break-before-make: primary should be off
AssertFalse(
	Condition := iDiscreteComponent.P_DiscreteStatus.PrimaryOutput,
	Message := 'Primary output should be FALSE during alternate state'
);

TEST_FINISHED();
END_METHOD

METHOD PRIVATE Test_DirectTransition_AlternateToActive
TEST(__POUNAME());

iDiscreteComponent := _GetDiscreteComponent(INDEX_ALTERNATE_TO_ACTIVE);
IF iDiscreteComponent = 0 THEN RETURN; END_IF
iDiscreteConfig := _GetDiscreteComponentConfig(INDEX_ALTERNATE_TO_ACTIVE);  // Same instance, different interface

// Skip this test for two-position devices
IF iDiscreteConfig.P_DiscreteConfiguration.PositionType = E_DiscretePositionType.TwoPositionDevice THEN
	TEST_FINISHED();
	RETURN;
END_IF

iDiscreteComponent.CyclicLogic();

// TODO: Start in Alternate state when command is available
// For now, manually set the secondary output
iDiscreteComponent.P_DiscreteStatus.SecondaryOutput := TRUE;
iDiscreteComponent.P_DiscreteStatus.PrimaryOutput := FALSE;
iDiscreteComponent.CyclicLogic();

AssertEquals_INT(
	Expected := TO_INT(E_DiscreteComponentState.Alternate),
	Actual := TO_INT(iDiscreteComponent.P_DiscreteStatus.BinaryComponentState),
	Message := 'Should start in Alternate state'
);

// Transition to Active
iDiscreteComponent.Activate();
iDiscreteComponent.P_DiscreteStatus.SecondaryOutput := FALSE;
iDiscreteComponent.P_DiscreteStatus.PrimaryOutput := TRUE;
iDiscreteComponent.CyclicLogic();

AssertEquals_INT(
	Expected := TO_INT(E_DiscreteComponentState.Active),
	Actual := TO_INT(iDiscreteComponent.P_DiscreteStatus.BinaryComponentState),
	Message := 'Should transition to Active state'
);

// Verify break-before-make: secondary should be off
AssertFalse(
	Condition := iDiscreteComponent.P_DiscreteStatus.SecondaryOutput,
	Message := 'Secondary output should be FALSE during active state'
);

TEST_FINISHED();
END_METHOD

METHOD PRIVATE Test_ErrorRecovery_ClearsAndReturnsToNeutral
TEST(__POUNAME());

iDiscreteComponent := _GetDiscreteComponent(INDEX_ERROR_RECOVERY);
IF iDiscreteComponent = 0 THEN RETURN; END_IF
iDiscreteComponent.CyclicLogic();

// Start in Active state
iDiscreteComponent.Activate();
iDiscreteComponent.CyclicLogic();

// TODO: Simulate error condition when error handling is implemented
// For now, test that deactivation from error clears outputs

// Deactivate to recover
iDiscreteComponent.Deactivate();
iDiscreteComponent.CyclicLogic();

AssertEquals_INT(
	Expected := TO_INT(E_DiscreteComponentState.Neutral),
	Actual := TO_INT(iDiscreteComponent.P_DiscreteStatus.BinaryComponentState),
	Message := 'Should return to Neutral state after error recovery'
);

AssertFalse(
	Condition := iDiscreteComponent.P_DiscreteStatus.PrimaryOutput,
	Message := 'Primary output should be cleared after recovery'
);

AssertFalse(
	Condition := iDiscreteComponent.P_DiscreteStatus.SecondaryOutput,
	Message := 'Secondary output should be cleared after recovery'
);

TEST_FINISHED();
END_METHOD

METHOD PRIVATE Test_InitializationSetsNeutralStateWithNoOutputs
TEST(__POUNAME());

iDiscreteComponent := _GetDiscreteComponent(INDEX_INITIALIZATION);
IF iDiscreteComponent = 0 THEN RETURN; END_IF

// Test pre-initialization state
AssertEquals_INT(
	Expected := TO_INT(E_DiscreteComponentState.Indeterminate),
	Actual := TO_INT(iDiscreteComponent.P_DiscreteStatus.BinaryComponentState),
	Message := 'Expected: Indeterminate starting state before initialization'
);

// Initialize and run one cycle
iDiscreteComponent.Initialize();
iDiscreteComponent.CyclicLogic();

// Test post-initialization state
AssertEquals_INT(
	Expected := TO_INT(E_DiscreteComponentState.Neutral),
	Actual := TO_INT(iDiscreteComponent.P_DiscreteStatus.BinaryComponentState),
	Message := 'Expected: Neutral state after initialization'
);

// Verify no outputs are active
AssertFalse(
	Condition := iDiscreteComponent.P_DiscreteStatus.PrimaryOutput,
	Message := 'Primary output should be FALSE after initialization'
);

AssertFalse(
	Condition := iDiscreteComponent.P_DiscreteStatus.SecondaryOutput,
	Message := 'Secondary output should be FALSE after initialization'
);

TEST_FINISHED();
END_METHOD

METHOD PRIVATE Test_InvalidCommand_DoesNotChangeOutputs
VAR
	savedPrimary : BOOL;
	savedSecondary : BOOL;
END_VAR
TEST(__POUNAME());

iDiscreteComponent := _GetDiscreteComponent(INDEX_INVALID_COMMAND);
IF iDiscreteComponent = 0 THEN RETURN; END_IF
iDiscreteComponent.CyclicLogic();

// Start in Active state
iDiscreteComponent.Activate();
iDiscreteComponent.CyclicLogic();

AssertEquals_INT(
	Expected := TO_INT(E_DiscreteComponentState.Active),
	Actual := TO_INT(iDiscreteComponent.P_DiscreteStatus.BinaryComponentState),
	Message := 'Should start in Active state'
);

// TODO: Send invalid command index when command system is fully implemented
// For now, test that invalid state transitions don't corrupt the state

// Save current state
savedPrimary := iDiscreteComponent.P_DiscreteStatus.PrimaryOutput;
savedSecondary := iDiscreteComponent.P_DiscreteStatus.SecondaryOutput;

// Try to execute command with invalid index (when implemented)
// fbComponent.ExecuteCommand(CmdIndex := 999);  // Invalid index
iDiscreteComponent.CyclicLogic();

// Outputs should remain unchanged
AssertEquals(
	Expected := savedPrimary,
	Actual := iDiscreteComponent.P_DiscreteStatus.PrimaryOutput,
	Message := 'Primary output should not change on invalid command'
);

AssertEquals(
	Expected := savedSecondary,
	Actual := iDiscreteComponent.P_DiscreteStatus.SecondaryOutput,
	Message := 'Secondary output should not change on invalid command'
);

TEST_FINISHED();
END_METHOD

METHOD PRIVATE Test_PermissiveInterlock_BlocksActivation
TEST(__POUNAME());

iDiscreteComponent := _GetDiscreteComponent(INDEX_INTERLOCK_ACTIVATION);
IF iDiscreteComponent = 0 THEN RETURN; END_IF
iDiscreteComponent.CyclicLogic();

// TODO: Implement when permissive interlock configuration is available
// Test that activation is blocked when interlock is not satisfied

// TODO: Implement when interlocks available
TEST_FINISHED();
END_METHOD

METHOD PRIVATE Test_PermissiveInterlock_BlocksAlternate
TEST(__POUNAME());

iDiscreteComponent := _GetDiscreteComponent(INDEX_INTERLOCK_ALTERNATE);
IF iDiscreteComponent = 0 THEN RETURN; END_IF
iDiscreteComponent.CyclicLogic();

// TODO: Implement when permissive interlock and alternate command are available
// Test that alternate activation is blocked when interlock is not satisfied

// TODO: Implement when interlocks available
TEST_FINISHED();
END_METHOD

METHOD PRIVATE Test_RapidStateChanges_EndInExpectedState
TEST(__POUNAME());

iDiscreteComponent := _GetDiscreteComponent(INDEX_RAPID_STATE_CHANGES);
IF iDiscreteComponent = 0 THEN RETURN; END_IF
iDiscreteComponent.CyclicLogic();

// Test rapid command sequence handling
// Note: Activate uses Monitored execution (continues running)
// Deactivate uses ImmediateEvaluation with higher priority

// Start from known state
iDiscreteComponent.Deactivate();
iDiscreteComponent.CyclicLogic();

// Issue Activate command
iDiscreteComponent.Activate();
iDiscreteComponent.CyclicLogic();

// Should be in Active state
AssertEquals_INT(
	Expected := TO_INT(E_DiscreteComponentState.Active),
	Actual := TO_INT(iDiscreteComponent.P_DiscreteStatus.BinaryComponentState),
	Message := 'Should be in Active state after Activate command'
);

// Deactivate with higher priority should override the Monitored Activate
iDiscreteComponent.Deactivate();
// Need extra cycle for command to be processed and override
iDiscreteComponent.CyclicLogic();

// With Monitored Activate still running but Deactivate having higher priority,
// the state depends on command system implementation
// Since Activate is Monitored and may still be executing, it could reactivate
AssertEquals_INT(
	Expected := TO_INT(E_DiscreteComponentState.Active),  // Monitored command still running
	Actual := TO_INT(iDiscreteComponent.P_DiscreteStatus.BinaryComponentState),
	Message := 'Monitored Activate may still be running after Deactivate'
);

// Clear all commands and test clean state changes
// Wait for any busy commands to complete
FOR i := 1 TO 10 DO
	iDiscreteComponent.CyclicLogic();
END_FOR

// Now test clean transitions
iDiscreteComponent.Deactivate();
iDiscreteComponent.CyclicLogic();
AssertEquals_INT(
	Expected := TO_INT(E_DiscreteComponentState.Neutral),
	Actual := TO_INT(iDiscreteComponent.P_DiscreteStatus.BinaryComponentState),
	Message := 'Should be Neutral after Deactivate with no other commands'
);

iDiscreteComponent.Activate();
iDiscreteComponent.CyclicLogic();
AssertEquals_INT(
	Expected := TO_INT(E_DiscreteComponentState.Active),
	Actual := TO_INT(iDiscreteComponent.P_DiscreteStatus.BinaryComponentState),
	Message := 'Should be Active after clean Activate'
);

TEST_FINISHED();
END_METHOD

METHOD PRIVATE Test_StateStabilityAcrossMultipleCycles
TEST(__POUNAME());

iDiscreteComponent := _GetDiscreteComponent(INDEX_STATE_STABILITY);
IF iDiscreteComponent = 0 THEN RETURN; END_IF
iDiscreteComponent.CyclicLogic();

// Test neutral state stability
FOR i := 1 TO 10 DO
	iDiscreteComponent.CyclicLogic();
END_FOR

AssertEquals_INT(
	Expected := TO_INT(E_DiscreteComponentState.Neutral),
	Actual := TO_INT(iDiscreteComponent.P_DiscreteStatus.BinaryComponentState),
	Message := 'Neutral state should remain stable across multiple cycles'
);

// Activate and test active state stability
iDiscreteComponent.Activate();
iDiscreteComponent.CyclicLogic();

FOR i := 1 TO 10 DO
	iDiscreteComponent.CyclicLogic();
END_FOR

AssertEquals_INT(
	Expected := TO_INT(E_DiscreteComponentState.Active),
	Actual := TO_INT(iDiscreteComponent.P_DiscreteStatus.BinaryComponentState),
	Message := 'Active state should remain stable across multiple cycles'
);

AssertTrue(
	Condition := iDiscreteComponent.P_DiscreteStatus.PrimaryOutput,
	Message := 'Primary output should remain TRUE during stable active state'
);

// Deactivate and test return to neutral stability
iDiscreteComponent.Deactivate();
iDiscreteComponent.CyclicLogic();

FOR i := 1 TO 10 DO
	iDiscreteComponent.CyclicLogic();
END_FOR

AssertEquals_INT(
	Expected := TO_INT(E_DiscreteComponentState.Neutral),
	Actual := TO_INT(iDiscreteComponent.P_DiscreteStatus.BinaryComponentState),
	Message := 'Should return to stable neutral state after deactivation'
);

TEST_FINISHED();
END_METHOD

METHOD PRIVATE Test_ThreePositionDevice_ActivatesAlternateOutputOnly
TEST(__POUNAME());

iDiscreteComponent := _GetDiscreteComponent(INDEX_THREE_POS_ALTERNATE);
IF iDiscreteComponent = 0 THEN RETURN; END_IF
iDiscreteConfig := _GetDiscreteComponentConfig(INDEX_THREE_POS_ALTERNATE);  // Same instance, different interface

// Skip this test for two-position devices
IF iDiscreteConfig.P_DiscreteConfiguration.PositionType = E_DiscretePositionType.TwoPositionDevice THEN
	TEST_FINISHED();
	RETURN;
END_IF

iDiscreteComponent.CyclicLogic();

// Test alternate/purge activation
// TODO: When alternate command is available, use it
// For now, manually set outputs

iDiscreteComponent.P_DiscreteStatus.PrimaryOutput := FALSE;
iDiscreteComponent.P_DiscreteStatus.SecondaryOutput := TRUE;
iDiscreteComponent.CyclicLogic();

AssertFalse(
	Condition := iDiscreteComponent.P_DiscreteStatus.PrimaryOutput,
	Message := 'Three-position device: primary output must be OFF in Alternate state'
);

AssertTrue(
	Condition := iDiscreteComponent.P_DiscreteStatus.SecondaryOutput,
	Message := 'Three-position device: secondary output should be ON for Alternate state'
);

AssertEquals_INT(
	Expected := TO_INT(E_DiscreteComponentState.Alternate),
	Actual := TO_INT(iDiscreteComponent.P_DiscreteStatus.BinaryComponentState),
	Message := 'Three-position device should be in Alternate state'
);

TEST_FINISHED();
END_METHOD

METHOD PRIVATE Test_ThreePositionDevice_ActivatesPrimaryOutputOnly
TEST(__POUNAME());

iDiscreteComponent := _GetDiscreteComponent(INDEX_THREE_POS_PRIMARY);
IF iDiscreteComponent = 0 THEN RETURN; END_IF
iDiscreteConfig := _GetDiscreteComponentConfig(INDEX_THREE_POS_PRIMARY);  // Same instance, different interface

// Skip this test for two-position devices
IF iDiscreteConfig.P_DiscreteConfiguration.PositionType = E_DiscretePositionType.TwoPositionDevice THEN
	TEST_FINISHED();
	RETURN;
END_IF

iDiscreteComponent.CyclicLogic();

// Three-position device: Neutral, Active (Vacuum), Alternate (Purge)
// Test primary activation

iDiscreteComponent.Activate();
iDiscreteComponent.CyclicLogic();

AssertTrue(
	Condition := iDiscreteComponent.P_DiscreteStatus.PrimaryOutput,
	Message := 'Three-position device: primary output should be ON for Active state'
);

AssertFalse(
	Condition := iDiscreteComponent.P_DiscreteStatus.SecondaryOutput,
	Message := 'Three-position device: secondary output must be OFF when primary is ON'
);

AssertEquals_INT(
	Expected := TO_INT(E_DiscreteComponentState.Active),
	Actual := TO_INT(iDiscreteComponent.P_DiscreteStatus.BinaryComponentState),
	Message := 'Three-position device should be in Active state'
);

TEST_FINISHED();
END_METHOD

METHOD PRIVATE Test_ThreePositionDevice_DeactivateTurnsOffBothOutputs
TEST(__POUNAME());

iDiscreteComponent := _GetDiscreteComponent(INDEX_THREE_POS_DEACTIVATE);
IF iDiscreteComponent = 0 THEN RETURN; END_IF
iDiscreteConfig := _GetDiscreteComponentConfig(INDEX_THREE_POS_DEACTIVATE);  // Same instance, different interface

// Skip this test for two-position devices
IF iDiscreteConfig.P_DiscreteConfiguration.PositionType = E_DiscretePositionType.TwoPositionDevice THEN
	TEST_FINISHED();
	RETURN;
END_IF

iDiscreteComponent.CyclicLogic();

// Test from Active state
iDiscreteComponent.Activate();
iDiscreteComponent.CyclicLogic();

iDiscreteComponent.Deactivate();
iDiscreteComponent.CyclicLogic();

AssertFalse(
	Condition := iDiscreteComponent.P_DiscreteStatus.PrimaryOutput,
	Message := 'Primary output should be OFF after deactivation from Active'
);

AssertFalse(
	Condition := iDiscreteComponent.P_DiscreteStatus.SecondaryOutput,
	Message := 'Secondary output should be OFF after deactivation'
);

// Test from Alternate state
iDiscreteComponent.P_DiscreteStatus.SecondaryOutput := TRUE;
iDiscreteComponent.CyclicLogic();

// Manually clear outputs to simulate deactivation (until command system is configured)
iDiscreteComponent.P_DiscreteStatus.PrimaryOutput := FALSE;
iDiscreteComponent.P_DiscreteStatus.SecondaryOutput := FALSE;
iDiscreteComponent.CyclicLogic();

AssertFalse(
	Condition := iDiscreteComponent.P_DiscreteStatus.PrimaryOutput,
	Message := 'Primary output should remain OFF'
);

AssertFalse(
	Condition := iDiscreteComponent.P_DiscreteStatus.SecondaryOutput,
	Message := 'Secondary output should be OFF after deactivation from Alternate'
);

AssertEquals_INT(
	Expected := TO_INT(E_DiscreteComponentState.Neutral),
	Actual := TO_INT(iDiscreteComponent.P_DiscreteStatus.BinaryComponentState),
	Message := 'Three-position device should return to Neutral from any state'
);

TEST_FINISHED();
END_METHOD

METHOD PRIVATE Test_ThreePositionDevice_NeverActivatesBothOutputsSimultaneously
TEST(__POUNAME());

iDiscreteComponent := _GetDiscreteComponent(INDEX_NEVER_BOTH_OUTPUTS);
IF iDiscreteComponent = 0 THEN RETURN; END_IF
iDiscreteConfig := _GetDiscreteComponentConfig(INDEX_NEVER_BOTH_OUTPUTS);  // Same instance, different interface

// Skip this test for two-position devices
IF iDiscreteConfig.P_DiscreteConfiguration.PositionType = E_DiscretePositionType.TwoPositionDevice THEN
	TEST_FINISHED();
	RETURN;
END_IF

iDiscreteComponent.CyclicLogic();

// Test 1: Activate primary output
iDiscreteComponent.Activate();
iDiscreteComponent.CyclicLogic();

AssertTrue(
	Condition := iDiscreteComponent.P_DiscreteStatus.PrimaryOutput,
	Message := 'Primary output should be TRUE when activated'
);

AssertFalse(
	Condition := iDiscreteComponent.P_DiscreteStatus.SecondaryOutput,
	Message := 'Secondary output must be FALSE when primary is active'
);

// Test 2: Try to manually force both outputs (simulating a fault condition)
// This should never happen in normal operation
iDiscreteComponent.P_DiscreteStatus.PrimaryOutput := TRUE;
iDiscreteComponent.P_DiscreteStatus.SecondaryOutput := TRUE;
iDiscreteComponent.CyclicLogic();

// The component should detect this as an invalid state
AssertEquals_INT(
	Expected := TO_INT(E_DiscreteComponentState.Alternate),  // Secondary takes priority per our logic
	Actual := TO_INT(iDiscreteComponent.P_DiscreteStatus.BinaryComponentState),
	Message := 'When both outputs are on, state should prioritize secondary (Alternate)'
);

// Test 3: Transition to alternate (when alternate command is available)
// For now, manually set outputs to test the protection
iDiscreteComponent.P_DiscreteStatus.PrimaryOutput := FALSE;
iDiscreteComponent.P_DiscreteStatus.SecondaryOutput := TRUE;
iDiscreteComponent.CyclicLogic();

AssertFalse(
	Condition := iDiscreteComponent.P_DiscreteStatus.PrimaryOutput,
	Message := 'Primary output must be FALSE when secondary is active'
);

AssertTrue(
	Condition := iDiscreteComponent.P_DiscreteStatus.SecondaryOutput,
	Message := 'Secondary output should be TRUE in alternate state'
);

// Verify state reflects alternate
AssertEquals_INT(
	Expected := TO_INT(E_DiscreteComponentState.Alternate),
	Actual := TO_INT(iDiscreteComponent.P_DiscreteStatus.BinaryComponentState),
	Message := 'State should be Alternate when only secondary output is active'
);

TEST_FINISHED();
END_METHOD

METHOD PRIVATE Test_TransitionFromActiveToAlternateTurnsOffActiveFirst
TEST(__POUNAME());

iDiscreteComponent := _GetDiscreteComponent(INDEX_BREAK_BEFORE_MAKE);
IF iDiscreteComponent = 0 THEN RETURN; END_IF
iDiscreteConfig := _GetDiscreteComponentConfig(INDEX_BREAK_BEFORE_MAKE);  // Same instance, different interface

// Skip this test for two-position devices
IF iDiscreteConfig.P_DiscreteConfiguration.PositionType = E_DiscretePositionType.TwoPositionDevice THEN
	TEST_FINISHED();
	RETURN;
END_IF

iDiscreteComponent.CyclicLogic();

// Step 1: Start with Active state (primary output on)
iDiscreteComponent.Activate();
iDiscreteComponent.CyclicLogic();

AssertTrue(
	Condition := iDiscreteComponent.P_DiscreteStatus.PrimaryOutput,
	Message := 'Primary output should be ON in Active state'
);

AssertFalse(
	Condition := iDiscreteComponent.P_DiscreteStatus.SecondaryOutput,
	Message := 'Secondary output should be OFF in Active state'
);

// Step 2: Transition to Alternate
// Since we don't have an Alternate command yet, we'll simulate the transition sequence
// CRITICAL: Primary must turn OFF before Secondary turns ON (break-before-make)

// First cycle: Turn off primary
iDiscreteComponent.P_DiscreteStatus.PrimaryOutput := FALSE;
iDiscreteComponent.CyclicLogic();

AssertFalse(
	Condition := iDiscreteComponent.P_DiscreteStatus.PrimaryOutput,
	Message := 'Primary output must be OFF during transition (break phase)'
);

AssertFalse(
	Condition := iDiscreteComponent.P_DiscreteStatus.SecondaryOutput,
	Message := 'Secondary output should still be OFF during break phase'
);

AssertEquals_INT(
	Expected := TO_INT(E_DiscreteComponentState.Neutral),
	Actual := TO_INT(iDiscreteComponent.P_DiscreteStatus.BinaryComponentState),
	Message := 'State should be Neutral when both outputs are off (transition phase)'
);

// Second cycle: Turn on secondary (after primary is confirmed off)
iDiscreteComponent.P_DiscreteStatus.SecondaryOutput := TRUE;
iDiscreteComponent.CyclicLogic();

AssertFalse(
	Condition := iDiscreteComponent.P_DiscreteStatus.PrimaryOutput,
	Message := 'Primary output must remain OFF when secondary is active'
);

AssertTrue(
	Condition := iDiscreteComponent.P_DiscreteStatus.SecondaryOutput,
	Message := 'Secondary output should be ON in Alternate state'
);

AssertEquals_INT(
	Expected := TO_INT(E_DiscreteComponentState.Alternate),
	Actual := TO_INT(iDiscreteComponent.P_DiscreteStatus.BinaryComponentState),
	Message := 'State should be Alternate after break-before-make transition'
);

// Step 3: Verify reverse transition (Alternate to Active) also uses break-before-make
iDiscreteComponent.P_DiscreteStatus.SecondaryOutput := FALSE;
iDiscreteComponent.CyclicLogic();

AssertEquals_INT(
	Expected := TO_INT(E_DiscreteComponentState.Neutral),
	Actual := TO_INT(iDiscreteComponent.P_DiscreteStatus.BinaryComponentState),
	Message := 'Should pass through Neutral state during reverse transition'
);

iDiscreteComponent.P_DiscreteStatus.PrimaryOutput := TRUE;
iDiscreteComponent.CyclicLogic();

AssertEquals_INT(
	Expected := TO_INT(E_DiscreteComponentState.Active),
	Actual := TO_INT(iDiscreteComponent.P_DiscreteStatus.BinaryComponentState),
	Message := 'State should return to Active after break-before-make reverse transition'
);

TEST_FINISHED();
END_METHOD

METHOD PRIVATE Test_TwoPositionDevice_ActivatesCorrectOutput
TEST(__POUNAME());

iDiscreteComponent := _GetDiscreteComponent(INDEX_TWO_POS_ACTIVATE);
IF iDiscreteComponent = 0 THEN RETURN; END_IF
iDiscreteComponent.CyclicLogic();

// Two-position device (e.g., simple on/off valve)
// Should only use primary output, never secondary

// Test activation
iDiscreteComponent.Activate();
iDiscreteComponent.CyclicLogic();

AssertTrue(
	Condition := iDiscreteComponent.P_DiscreteStatus.PrimaryOutput,
	Message := 'Two-position device should activate primary output'
);

AssertFalse(
	Condition := iDiscreteComponent.P_DiscreteStatus.SecondaryOutput,
	Message := 'Two-position device should never use secondary output'
);

AssertEquals_INT(
	Expected := TO_INT(E_DiscreteComponentState.Active),
	Actual := TO_INT(iDiscreteComponent.P_DiscreteStatus.BinaryComponentState),
	Message := 'Two-position device should be in Active state when on'
);

// Multiple activations should be idempotent
iDiscreteComponent.Activate();
iDiscreteComponent.CyclicLogic();

AssertTrue(
	Condition := iDiscreteComponent.P_DiscreteStatus.PrimaryOutput,
	Message := 'Primary output should remain TRUE after multiple activations'
);

TEST_FINISHED();
END_METHOD

METHOD PRIVATE Test_TwoPositionDevice_DeactivatesAllOutputs
TEST(__POUNAME());

iDiscreteComponent := _GetDiscreteComponent(INDEX_TWO_POS_DEACTIVATE);
IF iDiscreteComponent = 0 THEN RETURN; END_IF
iDiscreteComponent.CyclicLogic();

// Start with device activated
iDiscreteComponent.Activate();
iDiscreteComponent.CyclicLogic();

AssertTrue(
	Condition := iDiscreteComponent.P_DiscreteStatus.PrimaryOutput,
	Message := 'Primary output should be ON after activation'
);

// Test deactivation
iDiscreteComponent.Deactivate();
iDiscreteComponent.CyclicLogic();

AssertFalse(
	Condition := iDiscreteComponent.P_DiscreteStatus.PrimaryOutput,
	Message := 'Two-position device should deactivate primary output'
);

AssertFalse(
	Condition := iDiscreteComponent.P_DiscreteStatus.SecondaryOutput,
	Message := 'Secondary output should remain OFF (never used)'
);

AssertEquals_INT(
	Expected := TO_INT(E_DiscreteComponentState.Neutral),
	Actual := TO_INT(iDiscreteComponent.P_DiscreteStatus.BinaryComponentState),
	Message := 'Two-position device should be in Neutral state when off'
);

TEST_FINISHED();
END_METHOD

METHOD PRIVATE Test_TwoPositionDevice_IgnoresAlternateRequest
TEST(__POUNAME());

iDiscreteComponent := _GetDiscreteComponent(INDEX_TWO_POS_IGNORE_ALT);
IF iDiscreteComponent = 0 THEN RETURN; END_IF
iDiscreteConfig := _GetDiscreteComponentConfig(INDEX_TWO_POS_IGNORE_ALT);  // Same instance, different interface

// Skip this test for three-position devices
IF iDiscreteConfig.P_DiscreteConfiguration.PositionType <> E_DiscretePositionType.TwoPositionDevice THEN
	TEST_FINISHED();
	RETURN;
END_IF

iDiscreteComponent.CyclicLogic();

// Two-position devices should ignore alternate/purge commands
// They only support Active and Neutral states

iDiscreteComponent.Activate();
iDiscreteComponent.CyclicLogic();

// Try to force alternate state (should be ignored/invalid for 2-position)
// When alternate command is available, it should be ignored
// For two-position devices, the secondary output should always be false

// The _UpdateComponentStatus should force secondary to FALSE for two-position devices
AssertFalse(
	Condition := iDiscreteComponent.P_DiscreteStatus.SecondaryOutput,
	Message := 'Two-position device should always have secondary output FALSE'
);

// Should remain in Active state since primary is still ON
AssertEquals_INT(
	Expected := TO_INT(E_DiscreteComponentState.Active),
	Actual := TO_INT(iDiscreteComponent.P_DiscreteStatus.BinaryComponentState),
	Message := 'Two-position device should remain in Active state'
);

// Test that state remains Active even after multiple cycles
iDiscreteComponent.CyclicLogic();
iDiscreteComponent.CyclicLogic();

AssertEquals_INT(
	Expected := TO_INT(E_DiscreteComponentState.Active),
	Actual := TO_INT(iDiscreteComponent.P_DiscreteStatus.BinaryComponentState),
	Message := 'Two-position device state should be stable'
);

TEST_FINISHED();
END_METHOD

END_FUNCTION_BLOCK

// POUs/Tests/FB_ActuatorFeedbackTests
FUNCTION_BLOCK FB_ActuatorFeedbackTests EXTENDS FB_ActuatorBasicTests

VAR
	afbActuatorFeedback					: ARRAY[GC_Discrete.INDEX_TEST_MIN..GC_Discrete.INDEX_TEST_MAX] OF FB_TestActuatorFeedback;
END_VAR
VAR CONSTANT
	// Feedback-specific test indices (25-30)
	INDEX_FEEDBACK_EXTEND_EARLY			: DINT := 25;
	INDEX_FEEDBACK_RETRACT_EARLY		: DINT := 26;
	INDEX_FEEDBACK_EXTEND_TIMEOUT		: DINT := 27;
	INDEX_FEEDBACK_RETRACT_TIMEOUT		: DINT := 28;
END_VAR

// Run inherited base tests
SUPER^();

// Run feedback-specific tests
Test_FeedbackExtend_CompletesEarlyOnSensor();
Test_FeedbackRetract_CompletesEarlyOnSensor();
Test_FeedbackExtend_TimeoutWithoutSensor();
Test_FeedbackRetract_TimeoutWithoutSensor();

METHOD PROTECTED _GetDiscreteComponent : I_DiscreteBase
VAR_INPUT
	Index : DINT;
END_VAR
// Return the actuator feedback instance at the given index
_GetDiscreteComponent := afbActuatorFeedback[Index];
END_METHOD

METHOD PROTECTED _GetDiscreteComponentConfig : I_DiscreteBaseConfiguration
VAR_INPUT
	Index : DINT;
END_VAR
// Return the actuator feedback instance at the given index as configuration interface
_GetDiscreteComponentConfig := afbActuatorFeedback[Index];
END_METHOD

METHOD PRIVATE Test_FeedbackExtend_CompletesEarlyOnSensor
VAR
	CycleCount : DINT := 0;
END_VAR
TEST(__POUNAME());

iDiscreteComponent := _GetDiscreteComponent(INDEX_FEEDBACK_EXTEND_EARLY);
IF iDiscreteComponent = 0 THEN RETURN; END_IF
iDiscreteComponent.CyclicLogic();

// Configure sensor debounce for simulation with minimal delays
IF __ISVALIDREF(afbActuatorFeedback[INDEX_FEEDBACK_EXTEND_EARLY].P_I_SensorCfgExt) THEN
	afbActuatorFeedback[INDEX_FEEDBACK_EXTEND_EARLY].P_I_SensorCfgExt.P_DebounceConfiguration.BaseConfiguration.InSimulation := TRUE;
	afbActuatorFeedback[INDEX_FEEDBACK_EXTEND_EARLY].P_I_SensorCfgExt.P_DebounceConfiguration.tOnDelay := T#10MS;
	afbActuatorFeedback[INDEX_FEEDBACK_EXTEND_EARLY].P_I_SensorCfgExt.P_DebounceConfiguration.tOffDelay := T#10MS;
END_IF
IF __ISVALIDREF(afbActuatorFeedback[INDEX_FEEDBACK_EXTEND_EARLY].P_I_SensorCfgRet) THEN
	afbActuatorFeedback[INDEX_FEEDBACK_EXTEND_EARLY].P_I_SensorCfgRet.P_DebounceConfiguration.BaseConfiguration.InSimulation := TRUE;
	afbActuatorFeedback[INDEX_FEEDBACK_EXTEND_EARLY].P_I_SensorCfgRet.P_DebounceConfiguration.tOnDelay := T#10MS;
	afbActuatorFeedback[INDEX_FEEDBACK_EXTEND_EARLY].P_I_SensorCfgRet.P_DebounceConfiguration.tOffDelay := T#10MS;
END_IF

// Start from retracted position (sensor shows retracted)
IF __ISVALIDREF(afbActuatorFeedback[INDEX_FEEDBACK_EXTEND_EARLY].P_I_SensorRet) THEN
	afbActuatorFeedback[INDEX_FEEDBACK_EXTEND_EARLY].P_I_SensorRet.P_RawSignal := TRUE;
END_IF
IF __ISVALIDREF(afbActuatorFeedback[INDEX_FEEDBACK_EXTEND_EARLY].P_I_SensorExt) THEN
	afbActuatorFeedback[INDEX_FEEDBACK_EXTEND_EARLY].P_I_SensorExt.P_RawSignal := FALSE;
END_IF

// Execute extend command
iDiscreteComponent.Activate();
iDiscreteComponent.CyclicLogic();

// Command should be accepted and busy
AssertEquals_INT(
	Expected := TO_INT(Base.E_CommandResult.Accepted),
	Actual := TO_INT(iDiscreteComponent.P_DiscreteStatus.ComponentStatus.iLastCommand.P_CommandStatus.Result),
	Message := 'Expected: Extend command accepted'
);

AssertTrue(
	Condition := iDiscreteComponent.P_DiscreteStatus.ComponentStatus.iLastCommand.Busy,
	Message := 'Expected: Command busy after execute'
);

// Run a few cycles (simulate actuator moving)
FOR CycleCount := 1 TO 10 DO
	iDiscreteComponent.CyclicLogic();
END_FOR

// Simulate sensor feedback - actuator reached extended position
IF __ISVALIDREF(afbActuatorFeedback[INDEX_FEEDBACK_EXTEND_EARLY].P_I_SensorRet) THEN
	afbActuatorFeedback[INDEX_FEEDBACK_EXTEND_EARLY].P_I_SensorRet.P_RawSignal := FALSE;
END_IF
IF __ISVALIDREF(afbActuatorFeedback[INDEX_FEEDBACK_EXTEND_EARLY].P_I_SensorExt) THEN
	afbActuatorFeedback[INDEX_FEEDBACK_EXTEND_EARLY].P_I_SensorExt.P_RawSignal := TRUE;
END_IF

// Run cycles to process sensor feedback (debounce delay + processing)
FOR CycleCount := 1 TO 10 DO
	iDiscreteComponent.CyclicLogic();
END_FOR

// Command should complete with Ok result (early completion, not timeout)
AssertEquals_INT(
	Expected := TO_INT(Base.E_CommandResult.Ok),
	Actual := TO_INT(iDiscreteComponent.P_DiscreteStatus.ComponentStatus.iLastCommand.P_CommandStatus.Result),
	Message := 'Expected: Command completed with Ok (not RequestTimeout)'
);

AssertFalse(
	Condition := iDiscreteComponent.P_DiscreteStatus.ComponentStatus.iLastCommand.Busy,
	Message := 'Expected: Command not busy after sensor feedback'
);

// Verify completion happened well before 5-second timeout
AssertTrue(
	Condition := CycleCount < 100,  // Should complete in <<100 cycles (far less than 5 seconds)
	Message := 'Expected: Early completion on sensor feedback, not timeout'
);

TEST_FINISHED();
END_METHOD

METHOD PRIVATE Test_FeedbackExtend_TimeoutWithoutSensor
VAR
	CycleCount : DINT := 0;
	MaxCycles : DINT := 600;  // Allow enough cycles for 5-second timeout (at typical cycle time)
END_VAR
TEST(__POUNAME());

iDiscreteComponent := _GetDiscreteComponent(INDEX_FEEDBACK_EXTEND_TIMEOUT);
IF iDiscreteComponent = 0 THEN RETURN; END_IF
iDiscreteComponent.CyclicLogic();

// Configure sensor debounce for simulation with minimal delays
IF __ISVALIDREF(afbActuatorFeedback[INDEX_FEEDBACK_EXTEND_TIMEOUT].P_I_SensorCfgExt) THEN
	afbActuatorFeedback[INDEX_FEEDBACK_EXTEND_TIMEOUT].P_I_SensorCfgExt.P_DebounceConfiguration.BaseConfiguration.InSimulation := TRUE;
	afbActuatorFeedback[INDEX_FEEDBACK_EXTEND_TIMEOUT].P_I_SensorCfgExt.P_DebounceConfiguration.tOnDelay := T#10MS;
	afbActuatorFeedback[INDEX_FEEDBACK_EXTEND_TIMEOUT].P_I_SensorCfgExt.P_DebounceConfiguration.tOffDelay := T#10MS;
END_IF
IF __ISVALIDREF(afbActuatorFeedback[INDEX_FEEDBACK_EXTEND_TIMEOUT].P_I_SensorCfgRet) THEN
	afbActuatorFeedback[INDEX_FEEDBACK_EXTEND_TIMEOUT].P_I_SensorCfgRet.P_DebounceConfiguration.BaseConfiguration.InSimulation := TRUE;
	afbActuatorFeedback[INDEX_FEEDBACK_EXTEND_TIMEOUT].P_I_SensorCfgRet.P_DebounceConfiguration.tOnDelay := T#10MS;
	afbActuatorFeedback[INDEX_FEEDBACK_EXTEND_TIMEOUT].P_I_SensorCfgRet.P_DebounceConfiguration.tOffDelay := T#10MS;
END_IF

// Start from retracted position
IF __ISVALIDREF(afbActuatorFeedback[INDEX_FEEDBACK_EXTEND_TIMEOUT].P_I_SensorRet) THEN
	afbActuatorFeedback[INDEX_FEEDBACK_EXTEND_TIMEOUT].P_I_SensorRet.P_RawSignal := TRUE;
END_IF
IF __ISVALIDREF(afbActuatorFeedback[INDEX_FEEDBACK_EXTEND_TIMEOUT].P_I_SensorExt) THEN
	afbActuatorFeedback[INDEX_FEEDBACK_EXTEND_TIMEOUT].P_I_SensorExt.P_RawSignal := FALSE;
END_IF

// Execute extend command
iDiscreteComponent.Activate();
iDiscreteComponent.CyclicLogic();

// Command should be accepted and busy
AssertTrue(
	Condition := iDiscreteComponent.P_DiscreteStatus.ComponentStatus.iLastCommand.Busy,
	Message := 'Expected: Command busy after execute'
);

// Run cycles WITHOUT setting sensor feedback (simulate stuck actuator)
// Keep sensor at retracted position - extended sensor never triggers
WHILE (iDiscreteComponent.P_DiscreteStatus.ComponentStatus.iLastCommand.Busy) AND (CycleCount < MaxCycles) DO
	iDiscreteComponent.CyclicLogic();
	CycleCount := CycleCount + 1;
END_WHILE

// Command should timeout with RequestTimeout result
AssertEquals_INT(
	Expected := TO_INT(Base.E_CommandResult.RequestTimeout),
	Actual := TO_INT(iDiscreteComponent.P_DiscreteStatus.ComponentStatus.iLastCommand.P_CommandStatus.Result),
	Message := 'Expected: Command timeout (RequestTimeout) when sensor feedback not received'
);

AssertFalse(
	Condition := iDiscreteComponent.P_DiscreteStatus.ComponentStatus.iLastCommand.Busy,
	Message := 'Expected: Command not busy after timeout'
);

AssertTrue(
	Condition := iDiscreteComponent.P_DiscreteStatus.ComponentStatus.iLastCommand.P_CommandStatus.BaseStatus.Error,
	Message := 'Expected: Error flag set on timeout'
);

TEST_FINISHED();
END_METHOD

METHOD PRIVATE Test_FeedbackRetract_CompletesEarlyOnSensor
VAR
	CycleCount : DINT := 0;
END_VAR
TEST(__POUNAME());

iDiscreteComponent := _GetDiscreteComponent(INDEX_FEEDBACK_RETRACT_EARLY);
IF iDiscreteComponent = 0 THEN RETURN; END_IF
iDiscreteComponent.CyclicLogic();

// Configure sensor debounce for simulation with minimal delays
IF __ISVALIDREF(afbActuatorFeedback[INDEX_FEEDBACK_RETRACT_EARLY].P_I_SensorCfgExt) THEN
	afbActuatorFeedback[INDEX_FEEDBACK_RETRACT_EARLY].P_I_SensorCfgExt.P_DebounceConfiguration.BaseConfiguration.InSimulation := TRUE;
	afbActuatorFeedback[INDEX_FEEDBACK_RETRACT_EARLY].P_I_SensorCfgExt.P_DebounceConfiguration.tOnDelay := T#10MS;
	afbActuatorFeedback[INDEX_FEEDBACK_RETRACT_EARLY].P_I_SensorCfgExt.P_DebounceConfiguration.tOffDelay := T#10MS;
END_IF
IF __ISVALIDREF(afbActuatorFeedback[INDEX_FEEDBACK_RETRACT_EARLY].P_I_SensorCfgRet) THEN
	afbActuatorFeedback[INDEX_FEEDBACK_RETRACT_EARLY].P_I_SensorCfgRet.P_DebounceConfiguration.BaseConfiguration.InSimulation := TRUE;
	afbActuatorFeedback[INDEX_FEEDBACK_RETRACT_EARLY].P_I_SensorCfgRet.P_DebounceConfiguration.tOnDelay := T#10MS;
	afbActuatorFeedback[INDEX_FEEDBACK_RETRACT_EARLY].P_I_SensorCfgRet.P_DebounceConfiguration.tOffDelay := T#10MS;
END_IF

// Start from extended position (sensor shows extended)
IF __ISVALIDREF(afbActuatorFeedback[INDEX_FEEDBACK_RETRACT_EARLY].P_I_SensorExt) THEN
	afbActuatorFeedback[INDEX_FEEDBACK_RETRACT_EARLY].P_I_SensorExt.P_RawSignal := TRUE;
END_IF
IF __ISVALIDREF(afbActuatorFeedback[INDEX_FEEDBACK_RETRACT_EARLY].P_I_SensorRet) THEN
	afbActuatorFeedback[INDEX_FEEDBACK_RETRACT_EARLY].P_I_SensorRet.P_RawSignal := FALSE;
END_IF

// Execute retract command
iDiscreteComponent.Deactivate();
iDiscreteComponent.CyclicLogic();

// Command should be accepted and busy
AssertEquals_INT(
	Expected := TO_INT(Base.E_CommandResult.Accepted),
	Actual := TO_INT(iDiscreteComponent.P_DiscreteStatus.ComponentStatus.iLastCommand.P_CommandStatus.Result),
	Message := 'Expected: Retract command accepted'
);

AssertTrue(
	Condition := iDiscreteComponent.P_DiscreteStatus.ComponentStatus.iLastCommand.Busy,
	Message := 'Expected: Command busy after execute'
);

// Run a few cycles (simulate actuator moving)
FOR CycleCount := 1 TO 10 DO
	iDiscreteComponent.CyclicLogic();
END_FOR

// Simulate sensor feedback - actuator reached retracted position
IF __ISVALIDREF(afbActuatorFeedback[INDEX_FEEDBACK_RETRACT_EARLY].P_I_SensorExt) THEN
	afbActuatorFeedback[INDEX_FEEDBACK_RETRACT_EARLY].P_I_SensorExt.P_RawSignal := FALSE;
END_IF
IF __ISVALIDREF(afbActuatorFeedback[INDEX_FEEDBACK_RETRACT_EARLY].P_I_SensorRet) THEN
	afbActuatorFeedback[INDEX_FEEDBACK_RETRACT_EARLY].P_I_SensorRet.P_RawSignal := TRUE;
END_IF

// Run cycles to process sensor feedback (debounce delay + processing)
FOR CycleCount := 1 TO 10 DO
	iDiscreteComponent.CyclicLogic();
END_FOR

// Command should complete with Ok result (early completion, not timeout)
AssertEquals_INT(
	Expected := TO_INT(Base.E_CommandResult.Ok),
	Actual := TO_INT(iDiscreteComponent.P_DiscreteStatus.ComponentStatus.iLastCommand.P_CommandStatus.Result),
	Message := 'Expected: Command completed with Ok (not RequestTimeout)'
);

AssertFalse(
	Condition := iDiscreteComponent.P_DiscreteStatus.ComponentStatus.iLastCommand.Busy,
	Message := 'Expected: Command not busy after sensor feedback'
);

// Verify completion happened well before 5-second timeout
AssertTrue(
	Condition := CycleCount < 100,  // Should complete in <<100 cycles (far less than 5 seconds)
	Message := 'Expected: Early completion on sensor feedback, not timeout'
);

TEST_FINISHED();
END_METHOD

METHOD PRIVATE Test_FeedbackRetract_TimeoutWithoutSensor
VAR
	CycleCount : DINT := 0;
	MaxCycles : DINT := 600;  // Allow enough cycles for 5-second timeout (at typical cycle time)
END_VAR
TEST(__POUNAME());

iDiscreteComponent := _GetDiscreteComponent(INDEX_FEEDBACK_RETRACT_TIMEOUT);
IF iDiscreteComponent = 0 THEN RETURN; END_IF
iDiscreteComponent.CyclicLogic();

// Configure sensor debounce for simulation with minimal delays
IF __ISVALIDREF(afbActuatorFeedback[INDEX_FEEDBACK_RETRACT_TIMEOUT].P_I_SensorCfgExt) THEN
	afbActuatorFeedback[INDEX_FEEDBACK_RETRACT_TIMEOUT].P_I_SensorCfgExt.P_DebounceConfiguration.BaseConfiguration.InSimulation := TRUE;
	afbActuatorFeedback[INDEX_FEEDBACK_RETRACT_TIMEOUT].P_I_SensorCfgExt.P_DebounceConfiguration.tOnDelay := T#10MS;
	afbActuatorFeedback[INDEX_FEEDBACK_RETRACT_TIMEOUT].P_I_SensorCfgExt.P_DebounceConfiguration.tOffDelay := T#10MS;
END_IF
IF __ISVALIDREF(afbActuatorFeedback[INDEX_FEEDBACK_RETRACT_TIMEOUT].P_I_SensorCfgRet) THEN
	afbActuatorFeedback[INDEX_FEEDBACK_RETRACT_TIMEOUT].P_I_SensorCfgRet.P_DebounceConfiguration.BaseConfiguration.InSimulation := TRUE;
	afbActuatorFeedback[INDEX_FEEDBACK_RETRACT_TIMEOUT].P_I_SensorCfgRet.P_DebounceConfiguration.tOnDelay := T#10MS;
	afbActuatorFeedback[INDEX_FEEDBACK_RETRACT_TIMEOUT].P_I_SensorCfgRet.P_DebounceConfiguration.tOffDelay := T#10MS;
END_IF

// Start from extended position
IF __ISVALIDREF(afbActuatorFeedback[INDEX_FEEDBACK_RETRACT_TIMEOUT].P_I_SensorExt) THEN
	afbActuatorFeedback[INDEX_FEEDBACK_RETRACT_TIMEOUT].P_I_SensorExt.P_RawSignal := TRUE;
END_IF
IF __ISVALIDREF(afbActuatorFeedback[INDEX_FEEDBACK_RETRACT_TIMEOUT].P_I_SensorRet) THEN
	afbActuatorFeedback[INDEX_FEEDBACK_RETRACT_TIMEOUT].P_I_SensorRet.P_RawSignal := FALSE;
END_IF

// Execute retract command
iDiscreteComponent.Deactivate();
iDiscreteComponent.CyclicLogic();

// Command should be accepted and busy
AssertTrue(
	Condition := iDiscreteComponent.P_DiscreteStatus.ComponentStatus.iLastCommand.Busy,
	Message := 'Expected: Command busy after execute'
);

// Run cycles WITHOUT setting sensor feedback (simulate stuck actuator)
// Keep sensor at extended position - retracted sensor never triggers
WHILE (iDiscreteComponent.P_DiscreteStatus.ComponentStatus.iLastCommand.Busy) AND (CycleCount < MaxCycles) DO
	iDiscreteComponent.CyclicLogic();
	CycleCount := CycleCount + 1;
END_WHILE

// Command should timeout with RequestTimeout result
AssertEquals_INT(
	Expected := TO_INT(Base.E_CommandResult.RequestTimeout),
	Actual := TO_INT(iDiscreteComponent.P_DiscreteStatus.ComponentStatus.iLastCommand.P_CommandStatus.Result),
	Message := 'Expected: Command timeout (RequestTimeout) when sensor feedback not received'
);

AssertFalse(
	Condition := iDiscreteComponent.P_DiscreteStatus.ComponentStatus.iLastCommand.Busy,
	Message := 'Expected: Command not busy after timeout'
);

AssertTrue(
	Condition := iDiscreteComponent.P_DiscreteStatus.ComponentStatus.iLastCommand.P_CommandStatus.BaseStatus.Error,
	Message := 'Expected: Error flag set on timeout'
);

TEST_FINISHED();
END_METHOD

END_FUNCTION_BLOCK

// POUs/Tests/FB_ElectrostaticTests
FUNCTION_BLOCK FB_ElectrostaticTests EXTENDS FB_DiscreteBaseTests

VAR
	afbElectrostatic 	: ARRAY[GC_Discrete.INDEX_TEST_MIN..GC_Discrete.INDEX_TEST_MAX] OF FB_Electrostatic;
END_VAR

// All test methods are inherited from FB_DiscreteBaseTests
SUPER^();

METHOD PROTECTED _GetDiscreteComponent : I_DiscreteBase
VAR_INPUT
	Index : DINT;
END_VAR
// Return the electrostatic instance at the given index
_GetDiscreteComponent := afbElectrostatic[Index];
END_METHOD

METHOD PROTECTED _GetDiscreteComponentConfig : I_DiscreteBaseConfiguration
VAR_INPUT
	Index : DINT;
END_VAR
// Return the electrostatic instance at the given index as configuration interface
_GetDiscreteComponentConfig := afbElectrostatic[Index];
END_METHOD

END_FUNCTION_BLOCK

// POUs/FB_Electrostatic
{attribute 'no_explicit_call' := 'do not call this POU directly'}
FUNCTION_BLOCK FB_Electrostatic EXTENDS FB_DiscreteBase
VAR CONSTANT
	INDEX_CMD_ON			: DINT := 0;
	INDEX_CMD_OFF			: DINT := 1;
END_VAR

METHOD Activate : Base.E_CommandResult
ExecuteCommand(CmdIndex := INDEX_CMD_ON);

IF SUPER^.iCommands[INDEX_CMD_ON].P_CommandStatus.Result = Base.E_CommandResult.Accepted THEN
	SUPER^._Activate();
END_IF

Activate := SUPER^.iCommands[INDEX_CMD_ON].P_CommandStatus.Result;
END_METHOD

METHOD Deactivate : Base.E_CommandResult
ExecuteCommand(CmdIndex := INDEX_CMD_OFF);

IF SUPER^.iCommands[INDEX_CMD_OFF].P_CommandStatus.Result = Base.E_CommandResult.Accepted THEN
	SUPER^._Deactivate();
END_IF

Deactivate := SUPER^.iCommands[INDEX_CMD_OFF].P_CommandStatus.Result;
END_METHOD

METHOD CyclicLogic
SUPER^.CyclicLogic();
END_METHOD

END_FUNCTION_BLOCK

// POUs/Tests/FB_VacuumPurgeTests
FUNCTION_BLOCK FB_VacuumPurgeTests EXTENDS FB_DiscreteBaseTests

VAR
	afbVacuumPurge		: ARRAY[GC_Discrete.INDEX_TEST_MIN..GC_Discrete.INDEX_TEST_MAX] OF FB_VacuumPurge;
END_VAR

// All test methods are inherited from FB_DiscreteBaseTests
SUPER^();

METHOD PROTECTED _GetDiscreteComponent : I_DiscreteBase
VAR_INPUT
	Index : DINT;
END_VAR
// Return the vacuum purge instance at the given index
_GetDiscreteComponent := afbVacuumPurge[Index];
END_METHOD

METHOD PROTECTED _GetDiscreteComponentConfig : I_DiscreteBaseConfiguration
VAR_INPUT
	Index : DINT;
END_VAR
// Return the vacuum purge instance at the given index as configuration interface
_GetDiscreteComponentConfig := afbVacuumPurge[Index];
END_METHOD

END_FUNCTION_BLOCK

// POUs/FB_VacuumPurge
{attribute 'no_explicit_call' := 'do not call this POU directly'}
FUNCTION_BLOCK FB_VacuumPurge EXTENDS FB_DiscreteBase
VAR CONSTANT
	INDEX_CMD_VAC			: DINT := 0;
	INDEX_CMD_PURGE			: DINT := 1;
END_VAR

METHOD Activate : Base.E_CommandResult
ExecuteCommand(CmdIndex := INDEX_CMD_VAC);

IF SUPER^.iCommands[INDEX_CMD_VAC].P_CommandStatus.Result = Base.E_CommandResult.Accepted THEN
	SUPER^._Activate();
END_IF

Activate := SUPER^.iCommands[INDEX_CMD_VAC].P_CommandStatus.Result;
END_METHOD

METHOD Deactivate : Base.E_CommandResult
ExecuteCommand(CmdIndex := INDEX_CMD_PURGE);

IF SUPER^.iCommands[INDEX_CMD_PURGE].P_CommandStatus.Result = Base.E_CommandResult.Accepted THEN
	SUPER^._Deactivate();
END_IF

Deactivate := SUPER^.iCommands[INDEX_CMD_PURGE].P_CommandStatus.Result;
END_METHOD

METHOD CyclicLogic
SUPER^.CyclicLogic();
END_METHOD

METHOD Purge : Base.E_CommandResult
// Alias for Deactivate (Purge turns off vacuum)
Purge := Deactivate();
END_METHOD

METHOD Vacuum : Base.E_CommandResult
// Alias for Activate (Vacuum is the active state)
Vacuum := Activate();
END_METHOD

END_FUNCTION_BLOCK

// POUs/MAIN
PROGRAM MAIN
VAR
	Electrostatic			: FB_Electrostatic;
	VacPurge				: FB_VacuumPurge;
	Actuator				: FB_Actuator;
	
	ExtendCmd				: BOOL;
	RetractCmd				: BOOL;
	
	ElectostaticActivate	: BOOL;
	TurnOnVacuum			: BOOL;
END_VAR

Electrostatic.CyclicLogic();
VacPurge.CyclicLogic();
Actuator.CyclicLogic();

IF ExtendCmd THEN
	Actuator.Extend();
	ExtendCmd := FALSE;
END_IF

IF RetractCmd THEN
	Actuator.Retract();
	RetractCmd := FALSE;
END_IF

IF ElectostaticActivate THEN
	Electrostatic.Activate();
	ElectostaticActivate := FALSE;
END_IF

IF TurnOnVacuum THEN
	VacPurge.Activate();
	TurnOnVacuum	:= FALSE;
END_IF

END_PROGRAM

// POUs/PRG_TEST
PROGRAM PRG_TEST
VAR
	VacuumPurgeTests		: FB_VacuumPurgeTests;
	ElectrostaticTests		: FB_ElectrostaticTests;
	ActuatorTests			: FB_ActuatorBasicTests;
	ActuatorFeedbackTests	: FB_ActuatorFeedbackTests;
END_VAR

TcUnit.RUN();

END_PROGRAM
